            AXIS_10_POSITION : Real;   // AXIS 10 POSITION
            AXIS_11_POSITION : Real;   // AXIS 11 POSITION
            AXIS_12_POSITION : Real;   // AXIS 12 POSITION
            AXIS_13_POSITION : Real;   // AXIS 13 POSITION
            AXIS_14_POSITION : Real;   // AXIS 14 POSITION
            AXIS_15_POSITION : Real;   // AXIS 15 POSITION
            AXIS_16_POSITION : Real;   // AXIS 16 POSITION
            AXIS_17_POSITION : Real;   // AXIS 17 POSITION
            AXIS_18_POSITION : Real;   // AXIS 18 POSITION
            AXIS_19_POSITION : Real;   // AXIS 19 POSITION
            AXIS_20_POSITION : Real;   // AXIS 20 POSITION
            AXIS_21_POSITION : Real;   // AXIS 21 POSITION
            AXIS_22_POSITION : Real;   // AXIS 22 POSITION
            AXIS_23_POSITION : Real;   // AXIS 23 POSITION
            AXIS_24_POSITION : Real;   // AXIS 24 POSITION
            AXIS_25_POSITION : Real;   // AXIS 25 POSITION
            AXIS_26_POSITION : Real;   // AXIS 26 POSITION
            AXIS_27_POSITION : Real;   // AXIS 27 POSITION
            AXIS_28_POSITION : Real;   // AXIS 28 POSITION
            AXIS_29_POSITION : Real;   // AXIS 29 POSITION
            AXIS_30_POSITION : Real;   // AXIS 30 POSITION
            AXIS_31_POSITION : Real;   // AXIS 31 POSITION
         END_STRUCT;
         AUX : Struct
            AUX1 : Bool;   // AUXILIAR 1
            AUX2 : Bool;   // AUXILIAR 2
            AUX3 : Bool;   // AUXILIAR 3
            AUX4 : Bool;   // AUXILIAR 4
            AUX5 : Bool;   // AUXILIAR 5
            AUX6 : Bool;   // AUXILIAR 6
            AUX7 : Bool;   // AUXILIAR 7
            AUX8 : Byte;   // AUXILIAR 8
            AUX9 : Byte;   // AUXILIAR 9
            AUX10 : Byte;   // AUXILIAR 10
            AUX11 : Byte;   // AUXILIAR 11
            AUX12 : Byte;   // AUXILIAR 12
            AUX13 : Byte;   // AUXILIAR 13
            AUX14 : Byte;   // AUXILIAR 14
         END_STRUCT;
         REFERENCE_SCREEN : Struct
            AXIS_SELECTED : Int;   // REFERENCE SCREEN AXIS SELECTED
            MEMO_AXIS_SELECTED : Int;   // REFERENCE SCREEN MEMORIZED AXIS SELECTED
            SCREEN_SELECTED : Bool;   // REFERENCE SCREEN SCREEN SELECTED
            READ_DATA : Bool;   // REFERENCE SCREEN READ DATA
            WRITE_DATA : Bool;   // REFERENCE SCREEN WRITE DATA
            TIMER_READ : TP_TIME;   // READ TIMER
         END_STRUCT;
      END_STRUCT;
      MG7 : Struct
         GENERAL_BITS : Struct
            SCREEN_BA3_SELECTED : Bool;   // SCREEN BA3 SELECTED / GENERAL BITS SCREEN BA3 SELECTED
            SCREEN_NC_MANUAL_SELECTED : Bool;   // SCREEN NC MANUAL SELECTED / GENERAL BITS SCREEN NC MANUAL SELECTED
            SCREEN_EB_MODE_SELECT : Bool;   // SCREEN EB MODE SELECT / GENERAL BITS SCREEN EB MODE SELECT
            SP0_3 : Bool;   // GENERAL BITS
            BA3_SELECTED_UNIT_1 : Bool;   // BA3 SELECTED UNIT 1 / GENERAL BITS BA3 LIST SELECTED UNIT 1
            BA3_SELECTED_UNIT_2 : Bool;   // BA3 SELECTED UNIT 2 / GENERAL BITS BA3 LIST SELECTED UNIT 2
            BA3_SELECTED_UNIT_3 : Bool;   // BA3 SELECTED UNIT 3 / GENERAL BITS BA3 LIST SELECTED UNIT 3
            BA3_SELECTED_UNIT_4 : Bool;   // BA3 SELECTED UNIT 4 / GENERAL BITS BA3 LIST SELECTED UNIT 4
            SP1_0 : Bool;   // TWO UNITS OPTION ENABLE / GENERAL BITS
            SPNDLS_SBH_SG_AUX : Bool;   // GENERAL BITS SPINDLES SBH SG AUX
            SPNDLS_SBH_SG_PULSE : Bool;   // GENERAL BITS SPINDLES SBH SG PULSE
            PLC_LINE_AXES_BYTE : Byte;   // GENERAL BITS PLC LINE AXES BYTE
            PLC_LINE_SPINDLES_BYTE : Byte;   // GENERAL BITS PLC LINE SPINDLES BYTE
            PLC_LINE_AXES : Int;   // GENERAL BITS PLC LINE AXES
            PLC_LINE_SPINDLES : Int;   // GENERAL BITS PLC LINE SPINDLES
            BA3_LIST : Int;   // GENERAL BITS BA3 LIST
            MINUS_KEY : Byte;   // GENERAL BITS MINUS KEY
            PLUS_KEY : Byte;   // GENERAL BITS PLUS KEY
         END_STRUCT;
         NC_AXES : Struct
            SOFTKEYS : Struct   // NC AXES SOFTKEYS
               LEFT : Struct
                  MANUAL_MODE : Bool;   // MANUAL MODE (CN-AXES SCREEN) / NC AXES SOFTKEYS MANUAL MODE
                  SEMIAUTOMATIC_MODE : Bool;   // SEMIAUTOMATIC MODE (CN-AXES SCREEN) / NC AXES SOFTKEYS SEMIAUTOMATIC MODE
                  REFERENCE_MODE : Bool;   // REFERENCE MODE (CN-AXES SCREEN) / NC AXES SOFTKEYS REFERENCE MODE
                  JOG_MODE : Bool;   // NC AXES SOFTKEYS SPARE
                  SPINDLES_SBH_SG : Bool;   // SPINDLES SBH SG (CN-AXES SCREEN) / NC AXES SOFTKEYS SPINDLES SBH SG
                  CONTINUOS_INCREMENTAL : Bool;   // CONTINUOS-INCREMENTAL (CN-AXES SCREEN) / NC AXES SOFTKEYS CONTINUOS INCREMENTAL
                  SP0_6 : Bool;   // NC AXES SOFTKEYS SP0 6
                  SP0_7 : Bool;   // NC AXES SOFTKEYS SP0 7
               END_STRUCT;
               RIGHT : Struct
                  JOG_PLUS : Bool;   // JOG PLUS (CN-AXES SCREEN) / NC AXES SOFTKEYS JOG PLUS
                  JOG_MINUS : Bool;   // JOG MINUS (CN-AXES SCREEN) / NC AXES SOFTKEYS JOG MINUS
                  BLOCK_DEVICE : Bool;   // BLOCK DEVICE (CN-AXES SCREEN) / NC AXES SOFTKEYS BLOCK DEVICE
                  UNBLOCK_DEVICE : Bool;   // UNBLOCK DEVICE (CN-AXES SCREEN) / NC AXES SOFTKEYS UNBLOCK DEVICE
                  SP1_4 : Bool;   // NC AXES SOFTKEYS SP1 4
                  CHANGE_PANEL_CONTROL : Bool;   // CHANGE PANEL CONTROL (CN-AXES SCREEN) / NC AXES SOFTKEYS CHANGE PANEL CONTROL
                  SP1_6 : Bool;   // NC AXES SOFTKEYS SP1 6
                  SP1_7 : Bool;   // NC AXES SOFTKEYS SP1 7
               END_STRUCT;
            END_STRUCT;
            PBS : Struct   // NC AXES PBS
               MICRON : Bool;   // NC AXES PBS MICRON
               MICRONS_10 : Bool;   // NC AXES PBS MICRONS 10
               MICRONS_100 : Bool;   // NC AXES PBS MICRONS 100
               MILIMETER : Bool;   // NC AXES PBS MILIMETER
               SP0_4 : Bool;
               SP0_5 : Bool;
               SP0_6 : Bool;
               SP0_7 : Bool;
               SP1_0 : Bool;
               SP1_1 : Bool;
               SP1_2 : Bool;
               SP1_3 : Bool;
               SP1_4 : Bool;
               SP1_5 : Bool;
               SP1_6 : Bool;
               SP1_7 : Bool;
            END_STRUCT;
            SOFTKEY_LEDS : Struct   // NC AXES SOFTKEY LEDS
               MANUAL_MODE : Bool;   // MANUAL MODE (SOFTKEY LEDS) / NC AXES SOFTKEY LEDS MANUAL MODE
               ES_MODE : Bool;   // NC AXES SOFTKEY LEDS ES MODE
               REFERENCE_MODE : Bool;   // NC AXES SOFTKEY LEDS REFERENCE MODE
               SP0_3 : Bool;   // NC AXES SOFTKEY LEDS SP0 3
               SPINDLES_SBH_SG : Bool;   // NC AXES SOFTKEY LEDS SPINDLES SBH SG
               CONTINUOS_INCREMENTAL : Bool;   // NC AXES SOFTKEY LEDS CONTINUOS INCREMENTAL
               EB_MODE : Bool;   // NC AXES SOFTKEY LEDS EB MODE
               VK_MODE : Bool;   // NC AXES SOFTKEY LEDS VK MODE
               JOG_PLUS : Bool;   // NC AXES SOFTKEY LEDS JOG PLUS
               JOG_MINUS : Bool;   // NC AXES SOFTKEY LEDS JOG MINUS
               BLOCK_DEVICE : Bool;   // NC AXES SOFTKEY LEDS BLOCK DEVICE
               UNBLOCK_DEVICE : Bool;   // NC AXES SOFTKEY LEDS UNBLOCK DEVICE
               SP1_4 : Bool;   // NC AXES SOFTKEY LEDS SP1 4
               CHANGE_PANEL_CONTROL : Bool;   // NC AXES SOFTKEY LEDS CHANGE PANEL CONTROL
               SP1_6 : Bool;   // NC AXES SOFTKEY LEDS SP1 6
               SP1_7 : Bool;   // NC AXES SOFTKEY LEDS SP1 7
            END_STRUCT;
            PBS_LEDS : Struct   // NC AXES PBS LEDS
               MICRON : Bool;   // NC AXES PBS LEDS MICRON
               MICRONS_10 : Bool;   // NC AXES PBS LEDS MICRONS_10
               MICRONS_100 : Bool;   // NC AXES PBS LEDS MICRONS_100
               MILIMETER : Bool;   // NC AXES PBS LEDS MILIMETER
               SP0_4 : Bool;
               SP0_5 : Bool;
               SP0_6 : Bool;
               SP0_7 : Bool;
               SP1_0 : Bool;
               SP1_1 : Bool;
               SP1_2 : Bool;
               SP1_3 : Bool;
               SP1_4 : Bool;
               SP1_5 : Bool;
               SP1_6 : Bool;
               SP1_7 : Bool;
            END_STRUCT;
         END_STRUCT;
         BA3 : Struct
            SOFTKEYS : Struct   // BA3 SOFTKEYS
               AUTOMATIC_MODE : Bool;   // AUTOMATIC MODE (BA3) / BA3 SOFTKEYS AUTOMATIC MODE
               SINGLE_MODE : Bool;   // SINGLE CYCLE MODE (BA3) / BA3 SOFTKEYS SINGLE MODE
               SEMIAUTOMATIC_MODE : Bool;   // SEMIAUTOMATIC MODE (BA3) / BA3 SOFTKEYS SEMIAUTOMATIC MODE
               MANUAL_MODE : Bool;   // MANUAL MODE (BA3) / BA3 SOFTKEYS MANUAL MODE
               START : Bool;   // START (BA3) / BA3 SOFTKEYS START
               STOP : Bool;   // STOP (BA3) / BA3 SOFTKEYS STOP
               SPARE_2 : Bool;   // BA3 SOFTKEYS SP0 6
               SPARE : Bool;   // BA3 SOFTKEYS SP0 7
               SET_GOOD_PART : Bool;   // BA3 SOFTKEYS CLAMP FIXTURE 1
               UNCLAMP_F1 : Bool;   // BA3 SOFTKEYS UNCLAMP FIXTURE 1
               CLAMP_F2 : Bool;   // BA3 SOFTKEYS CLAMP FIXTURE 2
               UNCLAMP_F2 : Bool;   // BA3 SOFTKEYS UNCLAMP FIXTURE 2
               UNBLOCK_DEVICE : Bool;   // BA3 SOFTKEYS UNBLOCK DEVICE
               HOME : Bool;   // HOME (BA3) / BA3 SOFTKEYS HOME
               END_OF_CYCLE : Bool;   // BA3 SOFTKEYS END OF CYCLE
               CHANGE_PANEL_CONTROL : Bool;   // BA3 SOFTKEYS CHANGE PANEL
            END_STRUCT;
            PBS : Struct   // BA3 PBS
               MICRON : Bool;   // BA3 PBS MICRON
               MICRONS_10 : Bool;   // BA3 PBS MICRONS_10
               MICRONS_100 : Bool;   // BA3 PBS MICRONS_100
               MILIMETER : Bool;   // BA3 PBS MILIMETER
               SP0_4 : Bool;
               SP0_5 : Bool;
               SP0_6 : Bool;
               SP0_7 : Bool;
               SP1_0 : Bool;
               SP1_1 : Bool;
               SP1_2 : Bool;
               SP1_3 : Bool;
               SP1_4 : Bool;
               SP1_5 : Bool;
               SP1_6 : Bool;
               SP1_7 : Bool;
            END_STRUCT;
            SOFTKEY_LEDS : Struct   // BA3 SOFTKEY LEDS
               ER_MODE : Bool;   // BA3 SOFTKEY LEDS ER MODE
               ES_MODE : Bool;   // BA3 SOFTKEY LEDS ES MODE
               HOME : Bool;   // BA3 SOFTKEY LEDS HOME
               START : Bool;   // BA3 SOFTKEY LEDS START
               STOP : Bool;   // BA3 SOFTKEY LEDS STOP
               CONTINUOS_INCREMENTAL : Bool;   // BA3 SOFTKEY LEDS CONTINUOS INCREMENTAL
               SP0_6 : Bool;   // BA3 SOFTKEY LEDS SP0 6
               SP0_7 : Bool;   // BA3 SOFTKEY LEDS SP0 7
               JOG_PLUS : Bool;   // BA3 SOFTKEY LEDS JOG PLUS
               JOG_MINUS : Bool;   // BA3 SOFTKEY LEDS JOG MINUS
               UNBLOCK_DEVICE : Bool;   // BA3 SOFTKEY LEDS UNBLOCK DEVICE
               CLAMP_F1 : Bool;   // BA3 SOFTKEY LEDS CLAMP F1
               UNCLAMP_F1 : Bool;   // BA3 SOFTKEY LEDS UNCLAMP F1
               CLAMP_F2 : Bool;   // BA3 SOFTKEY LEDS CLAMP F2
               UNCLAMP_F2 : Bool;   // BA3 SOFTKEY LEDS UNCLAMP F2
               SP1_7 : Bool;   // BA3 SOFTKEY LEDS SP1 7
            END_STRUCT;
            PBS_LEDS : Struct   // BA3 PBS LEDS
               MICRON : Bool;   // BA3 PBS LEDS MICRON
               MICRONS_10 : Bool;   // BA3 PBS LEDS MICRONS_10
               MICRONS_100 : Bool;   // BA3 PBS LEDS MICRONS_100
               MILIMETER : Bool;   // BA3 PBS LEDS MILIMETER
               SP0_4 : Bool;
               SP0_5 : Bool;
               SP0_6 : Bool;
               SP0_7 : Bool;
               SP1_0 : Bool;
               SP1_1 : Bool;
               SP1_2 : Bool;
               SP1_3 : Bool;
               SP1_4 : Bool;
               SP1_5 : Bool;
               SP1_6 : Bool;
               BA3_MODE_SELECTED : Bool;
            END_STRUCT;
         END_STRUCT;
         AXIS_SELECTED : Struct
            AXIS_1_SELECTED : Bool;   // SPINDLE SP11 SELECTED / AXIS 1 SELECTED
            AXIS_2_SELECTED : Bool;   // SPINDLE SP12 SELECTED / AXIS 2 SELECTED
            AXIS_3_SELECTED : Bool;   // SPINDLE SP13 SELECTED / AXIS 3 SELECTED
            AXIS_4_SELECTED : Bool;   // SPINDLE SP14 SELECTED / AXIS 4 SELECTED
            AXIS_5_SELECTED : Bool;   // AXIS X1 SELECTED / AXIS 5 SELECTED
            AXIS_6_SELECTED : Bool;   // AXIS Y1 SELECTED / AXIS 6 SELECTED
            AXIS_7_SELECTED : Bool;   // AXIS Z11 SELECTED / AXIS 7 SELECTED
            AXIS_8_SELECTED : Bool;   // AXIS Z12 SELECTED / AXIS 8 SELECTED
            AXIS_9_SELECTED : Bool;   // AXIS X2 SELECTED / AXIS 9 SELECTED
            AXIS_10_SELECTED : Bool;   // AXIS Y2 SELECTED / AXIS 10 SELECTED
            AXIS_11_SELECTED : Bool;   // AXIS Z21 SELECTED / AXIS 11 SELECTED
            AXIS_12_SELECTED : Bool;   // AXIS Z22 SELECTED / AXIS 12 SELECTED
            AXIS_13_SELECTED : Bool;   // AXIS Q1 SELECTED / AXIS 13 SELECTED
            AXIS_14_SELECTED : Bool;   // AXIS Q2 SELECTED / AXIS 14 SELECTED
            AXIS_15_SELECTED : Bool;   // AXIS A1 SELECTED / AXIS 15 SELECTED
            AXIS_16_SELECTED : Bool;   // AXIS B SELECTED / AXIS 16 SELECTED
            AXIS_17_SELECTED : Bool;   // AXIS W SELECTED / AXIS 17 SELECTED
            AXIS_18_SELECTED : Bool;   // AXIS E SELECTED / AXIS 18 SELECTED
            AXIS_19_SELECTED : Bool;   // AXIS A2 SELECTED / AXIS 19 SELECTED
            AXIS_20_SELECTED : Bool;   // AXIS V1 SELECTED / AXIS 20 SELECTED
            AXIS_21_SELECTED : Bool;   // AXIS V2 SELECTED / AXIS 21 SELECTED
            AXIS_22_SELECTED : Bool;   // AXIS R SELECTED / AXIS 22 SELECTED
            AXIS_23_SELECTED : Bool;   // AXIS U1 SELECTED / AXIS 23 SELECTED
            AXIS_24_SELECTED : Bool;   // AXIS U2 SELECTED / AXIS 24 SELECTED
            AXIS_25_SELECTED : Bool;   // AXIS C SELECTED / AXIS 25 SELECTED
            AXIS_26_SELECTED : Bool;   // AXIS W1 SELECTED / AXIS 26 SELECTED
            AXIS_27_SELECTED : Bool;   // AXIS V SELECTED / AXIS 27 SELECTED
            AXIS_28_SELECTED : Bool;   // AXIS 28 SELECTED
            AXIS_29_SELECTED : Bool;   // AXIS 29 SELECTED
            AXIS_30_SELECTED : Bool;   // AXIS 30 SELECTED
            AXIS_31_SELECTED : Bool;   // AXIS 31 SELECTED
            SPARE_33_7 : Bool;   // SPARE_33_7
         END_STRUCT;
         AXIS_REFERENCED : Struct
            AXIS_1_REFERENCED : Bool;   // SPINDLE SP11 REFERENCED / AXIS 1 REFERENCED
            AXIS_2_REFERENCED : Bool;   // SPINDLE SP12 REFERENCED / AXIS 2 REFERENCED
            AXIS_3_REFERENCED : Bool;   // SPINDLE SP13 REFERENCED / AXIS 3 REFERENCED
            AXIS_4_REFERENCED : Bool;   // SPINDLE SP14 REFERENCED / AXIS 4 REFERENCED
            AXIS_5_REFERENCED : Bool;   // AXIS X1 REFERENCED / AXIS 5 REFERENCED
            AXIS_6_REFERENCED : Bool;   // AXIS Y1 REFERENCED / AXIS 6 REFERENCED
            AXIS_7_REFERENCED : Bool;   // AXIS Z11 REFERENCED / AXIS 7 REFERENCED
            AXIS_8_REFERENCED : Bool;   // AXIS Z12 REFERENCED / AXIS 8 REFERENCED
            AXIS_9_REFERENCED : Bool;   // AXIS X2 REFERENCED / AXIS 9 REFERENCED
            AXIS_10_REFERENCED : Bool;   // AXIS Y2 REFERENCED / AXIS 10 REFERENCED
            AXIS_11_REFERENCED : Bool;   // AXIS Z21 REFERENCED / AXIS 11 REFERENCED
            AXIS_12_REFERENCED : Bool;   // AXIS Z22 REFERENCED / AXIS 12 REFERENCED
            AXIS_13_REFERENCED : Bool;   // AXIS Q1 REFERENCED / AXIS 13 REFERENCED
            AXIS_14_REFERENCED : Bool;   // AXIS Q2 REFERENCED / AXIS 14 REFERENCED
            AXIS_15_REFERENCED : Bool;   // AXIS A1 REFERENCED / AXIS 15 REFERENCED
            AXIS_16_REFERENCED : Bool;   // AXIS B REFERENCED / AXIS 16 REFERENCED
            AXIS_17_REFERENCED : Bool;   // AXIS W REFERENCED / AXIS 17 REFERENCED
            AXIS_18_REFERENCED : Bool;   // AXIS E REFERENCED / AXIS 18 REFERENCED
            AXIS_19_REFERENCED : Bool;   // AXIS A2 REFERENCED / AXIS 19 REFERENCED
            AXIS_20_REFERENCED : Bool;   // AXIS V1 REFERENCED / AXIS 20 REFERENCED
            AXIS_21_REFERENCED : Bool;   // AXIS V2 REFERENCED / AXIS 21 REFERENCED
            AXIS_22_REFERENCED : Bool;   // AXIS R REFERENCED / AXIS 22 REFERENCED
            AXIS_23_REFERENCED : Bool;   // AXIS U1 REFERENCED / AXIS 23 REFERENCED
            AXIS_24_REFERENCED : Bool;   // AXIS U2 REFERENCED / AXIS 24 REFERENCED
            AXIS_25_REFERENCED : Bool;   // AXIS C REFERENCED / AXIS 25 REFERENCED
            AXIS_26_REFERENCED : Bool;   // AXIS W1 REFERENCED / AXIS 26 REFERENCED
            AXIS_27_REFERENCED : Bool;   // AXIS V REFERENCED / AXIS 27 REFERENCED
            AXIS_28_REFERENCED : Bool;   // AXIS 28 REFERENCED
            AXIS_29_REFERENCED : Bool;   // AXIS 29 REFERENCED
            AXIS_30_REFERENCED : Bool;   // AXIS 30 REFERENCED
            AXIS_31_REFERENCED : Bool;   // AXIS 31 REFERENCED
            SPARE_37_7 : Bool;   // SPARE_37_7
         END_STRUCT;
         AXIS_CONDITIONS : Struct
            AXIS_1_CONDITIONS : Bool;   // SPINDLE SP11 CONDITIONS / AXIS 1 CONDITIONS
            AXIS_2_CONDITIONS : Bool;   // SPINDLE SP12 CONDITIONS / AXIS 2 CONDITIONS
            AXIS_3_CONDITIONS : Bool;   // SPINDLE SP13 CONDITIONS / AXIS 3 CONDITIONS
            AXIS_4_CONDITIONS : Bool;   // SPINDLE SP14 CONDITIONS / AXIS 4 CONDITIONS
            AXIS_5_CONDITIONS : Bool;   // AXIS X1 CONDITIONS / AXIS 5 CONDITIONS
            AXIS_6_CONDITIONS : Bool;   // AXIS Y1 CONDITIONS / AXIS 6 CONDITIONS
            AXIS_7_CONDITIONS : Bool;   // AXIS Z11 CONDITIONS / AXIS 7 CONDITIONS
            AXIS_8_CONDITIONS : Bool;   // AXIS Z12 CONDITIONS / AXIS 8 CONDITIONS
            AXIS_9_CONDITIONS : Bool;   // AXIS X2 CONDITIONS / AXIS 9 CONDITIONS
            AXIS_10_CONDITIONS : Bool;   // AXIS Y2 CONDITIONS / AXIS 10 CONDITIONS
            AXIS_11_CONDITIONS : Bool;   // AXIS Z21 CONDITIONS / AXIS 11 CONDITIONS
            AXIS_12_CONDITIONS : Bool;   // AXIS Z22 CONDITIONS / AXIS 12 CONDITIONS
            AXIS_13_CONDITIONS : Bool;   // AXIS Q1 CONDITIONS / AXIS 13 CONDITIONS
            AXIS_14_CONDITIONS : Bool;   // AXIS Q2 CONDITIONS / AXIS 14 CONDITIONS
            AXIS_15_CONDITIONS : Bool;   // AXIS A1 CONDITIONS / AXIS 15 CONDITIONS
            AXIS_16_CONDITIONS : Bool;   // AXIS B CONDITIONS / AXIS 16 CONDITIONS
            AXIS_17_CONDITIONS : Bool;   // AXIS W CONDITIONS / AXIS 17 CONDITIONS
            AXIS_18_CONDITIONS : Bool;   // AXIS E CONDITIONS / AXIS 18 CONDITIONS
            AXIS_19_CONDITIONS : Bool;   // AXIS A2 CONDITIONS / AXIS 19 CONDITIONS
            AXIS_20_CONDITIONS : Bool;   // AXIS V1 CONDITIONS / AXIS 20 CONDITIONS
            AXIS_21_CONDITIONS : Bool;   // AXIS V2 CONDITIONS / AXIS 21 CONDITIONS
            AXIS_22_CONDITIONS : Bool;   // AXIS R CONDITIONS / AXIS 22 CONDITIONS
            AXIS_23_CONDITIONS : Bool;   // AXIS U1 CONDITIONS / AXIS 23 CONDITIONS
            AXIS_24_CONDITIONS : Bool;   // AXIS U2 CONDITIONS / AXIS 24 CONDITIONS
            AXIS_25_CONDITIONS : Bool;   // AXIS C CONDITIONS / AXIS 25 CONDITIONS
            AXIS_26_CONDITIONS : Bool;   // AXIS W1 CONDITIONS / AXIS 26 CONDITIONS
            AXIS_27_CONDITIONS : Bool;   // AXIS V CONDITIONS / AXIS 27 CONDITIONS
            AXIS_28_CONDITIONS : Bool;   // AXIS 28 CONDITIONS
            AXIS_29_CONDITIONS : Bool;   // AXIS 29 CONDITIONS
            AXIS_30_CONDITIONS : Bool;   // AXIS 30 CONDITIONS
            AXIS_31_CONDITIONS : Bool;   // AXIS 31 CONDITIONS
            SPARE_41_7 : Bool;   // SPARE_41_7
         END_STRUCT;
         AXIS_POSITION : Struct
            AXIS_1_POSITION : Real;   // AXIS 1 POSITION
            AXIS_2_POSITION : Real;   // AXIS 2 POSITION
            AXIS_3_POSITION : Real;   // AXIS 3 POSITION
            AXIS_4_POSITION : Real;   // AXIS 4 POSITION
            AXIS_5_POSITION : Real;   // AXIS 5 POSITION
            AXIS_6_POSITION : Real;   // AXIS 6 POSITION
            AXIS_7_POSITION : Real;   // AXIS 7 POSITION
            AXIS_8_POSITION : Real;   // AXIS 8 POSITION
            AXIS_9_POSITION : Real;   // AXIS 9 POSITION
            AXIS_10_POSITION : Real;   // AXIS 10 POSITION
            AXIS_11_POSITION : Real;   // AXIS 11 POSITION
            AXIS_12_POSITION : Real;   // AXIS 12 POSITION
            AXIS_13_POSITION : Real;   // AXIS 13 POSITION
            AXIS_14_POSITION : Real;   // AXIS 14 POSITION
            AXIS_15_POSITION : Real;   // AXIS 15 POSITION
            AXIS_16_POSITION : Real;   // AXIS 16 POSITION
            AXIS_17_POSITION : Real;   // AXIS 17 POSITION
            AXIS_18_POSITION : Real;   // AXIS 18 POSITION
            AXIS_19_POSITION : Real;   // AXIS 19 POSITION
            AXIS_20_POSITION : Real;   // AXIS 20 POSITION
            AXIS_21_POSITION : Real;   // AXIS 21 POSITION
            AXIS_22_POSITION : Real;   // AXIS 22 POSITION
            AXIS_23_POSITION : Real;   // AXIS 23 POSITION
            AXIS_24_POSITION : Real;   // AXIS 24 POSITION
            AXIS_25_POSITION : Real;   // AXIS 25 POSITION
            AXIS_26_POSITION : Real;   // AXIS 26 POSITION
            AXIS_27_POSITION : Real;   // AXIS 27 POSITION
            AXIS_28_POSITION : Real;   // AXIS 28 POSITION
            AXIS_29_POSITION : Real;   // AXIS 29 POSITION
            AXIS_30_POSITION : Real;   // AXIS 30 POSITION
            AXIS_31_POSITION : Real;   // AXIS 31 POSITION
         END_STRUCT;
         AUX : Struct
            AUX1 : Bool;   // AUXILIAR 1
            AUX2 : Bool;   // AUXILIAR 2
            AUX3 : Bool;   // AUXILIAR 3
            AUX4 : Bool;   // AUXILIAR 4
            AUX5 : Bool;   // AUXILIAR 5
            AUX6 : Bool;   // AUXILIAR 6
            AUX7 : Bool;   // AUXILIAR 7
            AUX8 : Byte;   // AUXILIAR 8
            AUX9 : Byte;   // AUXILIAR 9
            AUX10 : Byte;   // AUXILIAR 10
            AUX11 : Byte;   // AUXILIAR 11
            AUX12 : Byte;   // AUXILIAR 12
            AUX13 : Byte;   // AUXILIAR 13
            AUX14 : Byte;   // AUXILIAR 14
         END_STRUCT;
         REFERENCE_SCREEN : Struct
            AXIS_SELECTED : Int;   // REFERENCE SCREEN AXIS SELECTED
            MEMO_AXIS_SELECTED : Int;   // REFERENCE SCREEN MEMORIZED AXIS SELECTED
            SCREEN_SELECTED : Bool;   // REFERENCE SCREEN SCREEN SELECTED
            READ_DATA : Bool;   // REFERENCE SCREEN READ DATA
            WRITE_DATA : Bool;   // REFERENCE SCREEN WRITE DATA
            TIMER_READ : TP_TIME;   // READ TIMER
         END_STRUCT;
      END_STRUCT;
      MG8 : Struct
         GENERAL_BITS : Struct
            SCREEN_BA3_SELECTED : Bool;   // SCREEN BA3 SELECTED / GENERAL BITS SCREEN BA3 SELECTED
            SCREEN_NC_MANUAL_SELECTED : Bool;   // SCREEN NC MANUAL SELECTED / GENERAL BITS SCREEN NC MANUAL SELECTED
            SCREEN_EB_MODE_SELECT : Bool;   // SCREEN EB MODE SELECT / GENERAL BITS SCREEN EB MODE SELECT
            SP0_3 : Bool;   // GENERAL BITS
            BA3_SELECTED_UNIT_1 : Bool;   // BA3 SELECTED UNIT 1 / GENERAL BITS BA3 LIST SELECTED UNIT 1
            BA3_SELECTED_UNIT_2 : Bool;   // BA3 SELECTED UNIT 2 / GENERAL BITS BA3 LIST SELECTED UNIT 2
            BA3_SELECTED_UNIT_3 : Bool;   // BA3 SELECTED UNIT 3 / GENERAL BITS BA3 LIST SELECTED UNIT 3
            BA3_SELECTED_UNIT_4 : Bool;   // BA3 SELECTED UNIT 4 / GENERAL BITS BA3 LIST SELECTED UNIT 4
            SP1_0 : Bool;   // TWO UNITS OPTION ENABLE / GENERAL BITS
            SPNDLS_SBH_SG_AUX : Bool;   // GENERAL BITS SPINDLES SBH SG AUX
            SPNDLS_SBH_SG_PULSE : Bool;   // GENERAL BITS SPINDLES SBH SG PULSE
            PLC_LINE_AXES_BYTE : Byte;   // GENERAL BITS PLC LINE AXES BYTE
            PLC_LINE_SPINDLES_BYTE : Byte;   // GENERAL BITS PLC LINE SPINDLES BYTE
            PLC_LINE_AXES : Int;   // GENERAL BITS PLC LINE AXES
            PLC_LINE_SPINDLES : Int;   // GENERAL BITS PLC LINE SPINDLES
            BA3_LIST : Int;   // GENERAL BITS BA3 LIST
            MINUS_KEY : Byte;   // GENERAL BITS MINUS KEY
            PLUS_KEY : Byte;   // GENERAL BITS PLUS KEY
         END_STRUCT;
         NC_AXES : Struct
            SOFTKEYS : Struct   // NC AXES SOFTKEYS
               LEFT : Struct
                  MANUAL_MODE : Bool;   // MANUAL MODE (CN-AXES SCREEN) / NC AXES SOFTKEYS MANUAL MODE
                  SEMIAUTOMATIC_MODE : Bool;   // SEMIAUTOMATIC MODE (CN-AXES SCREEN) / NC AXES SOFTKEYS SEMIAUTOMATIC MODE
                  REFERENCE_MODE : Bool;   // REFERENCE MODE (CN-AXES SCREEN) / NC AXES SOFTKEYS REFERENCE MODE
                  JOG_MODE : Bool;   // NC AXES SOFTKEYS SPARE
                  SPINDLES_SBH_SG : Bool;   // SPINDLES SBH SG (CN-AXES SCREEN) / NC AXES SOFTKEYS SPINDLES SBH SG
                  CONTINUOS_INCREMENTAL : Bool;   // CONTINUOS-INCREMENTAL (CN-AXES SCREEN) / NC AXES SOFTKEYS CONTINUOS INCREMENTAL
                  SP0_6 : Bool;   // NC AXES SOFTKEYS SP0 6
                  SP0_7 : Bool;   // NC AXES SOFTKEYS SP0 7
               END_STRUCT;
               RIGHT : Struct
                  JOG_PLUS : Bool;   // JOG PLUS (CN-AXES SCREEN) / NC AXES SOFTKEYS JOG PLUS
                  JOG_MINUS : Bool;   // JOG MINUS (CN-AXES SCREEN) / NC AXES SOFTKEYS JOG MINUS
                  BLOCK_DEVICE : Bool;   // BLOCK DEVICE (CN-AXES SCREEN) / NC AXES SOFTKEYS BLOCK DEVICE
                  UNBLOCK_DEVICE : Bool;   // UNBLOCK DEVICE (CN-AXES SCREEN) / NC AXES SOFTKEYS UNBLOCK DEVICE
                  SP1_4 : Bool;   // NC AXES SOFTKEYS SP1 4
                  CHANGE_PANEL_CONTROL : Bool;   // CHANGE PANEL CONTROL (CN-AXES SCREEN) / NC AXES SOFTKEYS CHANGE PANEL CONTROL
                  SP1_6 : Bool;   // NC AXES SOFTKEYS SP1 6
                  SP1_7 : Bool;   // NC AXES SOFTKEYS SP1 7
               END_STRUCT;
            END_STRUCT;
            PBS : Struct   // NC AXES PBS
               MICRON : Bool;   // NC AXES PBS MICRON
               MICRONS_10 : Bool;   // NC AXES PBS MICRONS 10
               MICRONS_100 : Bool;   // NC AXES PBS MICRONS 100
               MILIMETER : Bool;   // NC AXES PBS MILIMETER
               SP0_4 : Bool;
               SP0_5 : Bool;
               SP0_6 : Bool;
               SP0_7 : Bool;
               SP1_0 : Bool;
               SP1_1 : Bool;
               SP1_2 : Bool;
               SP1_3 : Bool;
               SP1_4 : Bool;
               SP1_5 : Bool;
               SP1_6 : Bool;
               SP1_7 : Bool;
            END_STRUCT;
            SOFTKEY_LEDS : Struct   // NC AXES SOFTKEY LEDS
               MANUAL_MODE : Bool;   // MANUAL MODE (SOFTKEY LEDS) / NC AXES SOFTKEY LEDS MANUAL MODE
               ES_MODE : Bool;   // NC AXES SOFTKEY LEDS ES MODE
               REFERENCE_MODE : Bool;   // NC AXES SOFTKEY LEDS REFERENCE MODE
               SP0_3 : Bool;   // NC AXES SOFTKEY LEDS SP0 3
               SPINDLES_SBH_SG : Bool;   // NC AXES SOFTKEY LEDS SPINDLES SBH SG
               CONTINUOS_INCREMENTAL : Bool;   // NC AXES SOFTKEY LEDS CONTINUOS INCREMENTAL
               EB_MODE : Bool;   // NC AXES SOFTKEY LEDS EB MODE
               VK_MODE : Bool;   // NC AXES SOFTKEY LEDS VK MODE
               JOG_PLUS : Bool;   // NC AXES SOFTKEY LEDS JOG PLUS
               JOG_MINUS : Bool;   // NC AXES SOFTKEY LEDS JOG MINUS
               BLOCK_DEVICE : Bool;   // NC AXES SOFTKEY LEDS BLOCK DEVICE
               UNBLOCK_DEVICE : Bool;   // NC AXES SOFTKEY LEDS UNBLOCK DEVICE
               SP1_4 : Bool;   // NC AXES SOFTKEY LEDS SP1 4
               CHANGE_PANEL_CONTROL : Bool;   // NC AXES SOFTKEY LEDS CHANGE PANEL CONTROL
               SP1_6 : Bool;   // NC AXES SOFTKEY LEDS SP1 6
               SP1_7 : Bool;   // NC AXES SOFTKEY LEDS SP1 7
            END_STRUCT;
            PBS_LEDS : Struct   // NC AXES PBS LEDS
               MICRON : Bool;   // NC AXES PBS LEDS MICRON
               MICRONS_10 : Bool;   // NC AXES PBS LEDS MICRONS_10
               MICRONS_100 : Bool;   // NC AXES PBS LEDS MICRONS_100
               MILIMETER : Bool;   // NC AXES PBS LEDS MILIMETER
               SP0_4 : Bool;
               SP0_5 : Bool;
               SP0_6 : Bool;
               SP0_7 : Bool;
               SP1_0 : Bool;
               SP1_1 : Bool;
               SP1_2 : Bool;
               SP1_3 : Bool;
               SP1_4 : Bool;
               SP1_5 : Bool;
               SP1_6 : Bool;
               SP1_7 : Bool;
            END_STRUCT;
         END_STRUCT;
         BA3 : Struct
            SOFTKEYS : Struct   // BA3 SOFTKEYS
               AUTOMATIC_MODE : Bool;   // AUTOMATIC MODE (BA3) / BA3 SOFTKEYS AUTOMATIC MODE
               SINGLE_MODE : Bool;   // SINGLE CYCLE MODE (BA3) / BA3 SOFTKEYS SINGLE MODE
               SEMIAUTOMATIC_MODE : Bool;   // SEMIAUTOMATIC MODE (BA3) / BA3 SOFTKEYS SEMIAUTOMATIC MODE
               MANUAL_MODE : Bool;   // MANUAL MODE (BA3) / BA3 SOFTKEYS MANUAL MODE
               START : Bool;   // START (BA3) / BA3 SOFTKEYS START
               STOP : Bool;   // STOP (BA3) / BA3 SOFTKEYS STOP
               SPARE_2 : Bool;   // BA3 SOFTKEYS SP0 6
               SPARE : Bool;   // BA3 SOFTKEYS SP0 7
               SET_GOOD_PART : Bool;   // BA3 SOFTKEYS CLAMP FIXTURE 1
               UNCLAMP_F1 : Bool;   // BA3 SOFTKEYS UNCLAMP FIXTURE 1
               CLAMP_F2 : Bool;   // BA3 SOFTKEYS CLAMP FIXTURE 2
               UNCLAMP_F2 : Bool;   // BA3 SOFTKEYS UNCLAMP FIXTURE 2
               UNBLOCK_DEVICE : Bool;   // BA3 SOFTKEYS UNBLOCK DEVICE
               HOME : Bool;   // HOME (BA3) / BA3 SOFTKEYS HOME
               END_OF_CYCLE : Bool;   // BA3 SOFTKEYS END OF CYCLE
               CHANGE_PANEL_CONTROL : Bool;   // BA3 SOFTKEYS CHANGE PANEL
            END_STRUCT;
            PBS : Struct   // BA3 PBS
               MICRON : Bool;   // BA3 PBS MICRON
               MICRONS_10 : Bool;   // BA3 PBS MICRONS_10
               MICRONS_100 : Bool;   // BA3 PBS MICRONS_100
               MILIMETER : Bool;   // BA3 PBS MILIMETER
               SP0_4 : Bool;
               SP0_5 : Bool;
               SP0_6 : Bool;
               SP0_7 : Bool;
               SP1_0 : Bool;
               SP1_1 : Bool;
               SP1_2 : Bool;
               SP1_3 : Bool;
               SP1_4 : Bool;
               SP1_5 : Bool;
               SP1_6 : Bool;
               SP1_7 : Bool;
            END_STRUCT;
            SOFTKEY_LEDS : Struct   // BA3 SOFTKEY LEDS
               ER_MODE : Bool;   // BA3 SOFTKEY LEDS ER MODE
               ES_MODE : Bool;   // BA3 SOFTKEY LEDS ES MODE
               HOME : Bool;   // BA3 SOFTKEY LEDS HOME
               START : Bool;   // BA3 SOFTKEY LEDS START
               STOP : Bool;   // BA3 SOFTKEY LEDS STOP
               CONTINUOS_INCREMENTAL : Bool;   // BA3 SOFTKEY LEDS CONTINUOS INCREMENTAL
               SP0_6 : Bool;   // BA3 SOFTKEY LEDS SP0 6
               SP0_7 : Bool;   // BA3 SOFTKEY LEDS SP0 7
               JOG_PLUS : Bool;   // BA3 SOFTKEY LEDS JOG PLUS
               JOG_MINUS : Bool;   // BA3 SOFTKEY LEDS JOG MINUS
               UNBLOCK_DEVICE : Bool;   // BA3 SOFTKEY LEDS UNBLOCK DEVICE
               CLAMP_F1 : Bool;   // BA3 SOFTKEY LEDS CLAMP F1
               UNCLAMP_F1 : Bool;   // BA3 SOFTKEY LEDS UNCLAMP F1
               CLAMP_F2 : Bool;   // BA3 SOFTKEY LEDS CLAMP F2
               UNCLAMP_F2 : Bool;   // BA3 SOFTKEY LEDS UNCLAMP F2
               SP1_7 : Bool;   // BA3 SOFTKEY LEDS SP1 7
            END_STRUCT;
            PBS_LEDS : Struct   // BA3 PBS LEDS
               MICRON : Bool;   // BA3 PBS LEDS MICRON
               MICRONS_10 : Bool;   // BA3 PBS LEDS MICRONS_10
               MICRONS_100 : Bool;   // BA3 PBS LEDS MICRONS_100
               MILIMETER : Bool;   // BA3 PBS LEDS MILIMETER
               SP0_4 : Bool;
               SP0_5 : Bool;
               SP0_6 : Bool;
               SP0_7 : Bool;
               SP1_0 : Bool;
               SP1_1 : Bool;
               SP1_2 : Bool;
               SP1_3 : Bool;
               SP1_4 : Bool;
               SP1_5 : Bool;
               SP1_6 : Bool;
               BA3_MODE_SELECTED : Bool;
            END_STRUCT;
         END_STRUCT;
         AXIS_SELECTED : Struct
            AXIS_1_SELECTED : Bool;   // SPINDLE SP11 SELECTED / AXIS 1 SELECTED
            AXIS_2_SELECTED : Bool;   // SPINDLE SP12 SELECTED / AXIS 2 SELECTED
            AXIS_3_SELECTED : Bool;   // SPINDLE SP13 SELECTED / AXIS 3 SELECTED
            AXIS_4_SELECTED : Bool;   // SPINDLE SP14 SELECTED / AXIS 4 SELECTED
            AXIS_5_SELECTED : Bool;   // AXIS X1 SELECTED / AXIS 5 SELECTED
            AXIS_6_SELECTED : Bool;   // AXIS Y1 SELECTED / AXIS 6 SELECTED
            AXIS_7_SELECTED : Bool;   // AXIS Z11 SELECTED / AXIS 7 SELECTED
            AXIS_8_SELECTED : Bool;   // AXIS Z12 SELECTED / AXIS 8 SELECTED
            AXIS_9_SELECTED : Bool;   // AXIS X2 SELECTED / AXIS 9 SELECTED
            AXIS_10_SELECTED : Bool;   // AXIS Y2 SELECTED / AXIS 10 SELECTED
            AXIS_11_SELECTED : Bool;   // AXIS Z21 SELECTED / AXIS 11 SELECTED
            AXIS_12_SELECTED : Bool;   // AXIS Z22 SELECTED / AXIS 12 SELECTED
            AXIS_13_SELECTED : Bool;   // AXIS Q1 SELECTED / AXIS 13 SELECTED
            AXIS_14_SELECTED : Bool;   // AXIS Q2 SELECTED / AXIS 14 SELECTED
            AXIS_15_SELECTED : Bool;   // AXIS A1 SELECTED / AXIS 15 SELECTED
            AXIS_16_SELECTED : Bool;   // AXIS B SELECTED / AXIS 16 SELECTED
            AXIS_17_SELECTED : Bool;   // AXIS W SELECTED / AXIS 17 SELECTED
            AXIS_18_SELECTED : Bool;   // AXIS E SELECTED / AXIS 18 SELECTED
            AXIS_19_SELECTED : Bool;   // AXIS A2 SELECTED / AXIS 19 SELECTED
            AXIS_20_SELECTED : Bool;   // AXIS V1 SELECTED / AXIS 20 SELECTED
            AXIS_21_SELECTED : Bool;   // AXIS V2 SELECTED / AXIS 21 SELECTED
            AXIS_22_SELECTED : Bool;   // AXIS R SELECTED / AXIS 22 SELECTED
            AXIS_23_SELECTED : Bool;   // AXIS U1 SELECTED / AXIS 23 SELECTED
            AXIS_24_SELECTED : Bool;   // AXIS U2 SELECTED / AXIS 24 SELECTED
            AXIS_25_SELECTED : Bool;   // AXIS C SELECTED / AXIS 25 SELECTED
            AXIS_26_SELECTED : Bool;   // AXIS W1 SELECTED / AXIS 26 SELECTED
            AXIS_27_SELECTED : Bool;   // AXIS V SELECTED / AXIS 27 SELECTED
            AXIS_28_SELECTED : Bool;   // AXIS 28 SELECTED
            AXIS_29_SELECTED : Bool;   // AXIS 29 SELECTED
            AXIS_30_SELECTED : Bool;   // AXIS 30 SELECTED
            AXIS_31_SELECTED : Bool;   // AXIS 31 SELECTED
            SPARE_33_7 : Bool;   // SPARE_33_7
         END_STRUCT;
         AXIS_REFERENCED : Struct
            AXIS_1_REFERENCED : Bool;   // SPINDLE SP11 REFERENCED / AXIS 1 REFERENCED
            AXIS_2_REFERENCED : Bool;   // SPINDLE SP12 REFERENCED / AXIS 2 REFERENCED
            AXIS_3_REFERENCED : Bool;   // SPINDLE SP13 REFERENCED / AXIS 3 REFERENCED
            AXIS_4_REFERENCED : Bool;   // SPINDLE SP14 REFERENCED / AXIS 4 REFERENCED
            AXIS_5_REFERENCED : Bool;   // AXIS X1 REFERENCED / AXIS 5 REFERENCED
            AXIS_6_REFERENCED : Bool;   // AXIS Y1 REFERENCED / AXIS 6 REFERENCED
            AXIS_7_REFERENCED : Bool;   // AXIS Z11 REFERENCED / AXIS 7 REFERENCED
            AXIS_8_REFERENCED : Bool;   // AXIS Z12 REFERENCED / AXIS 8 REFERENCED
            AXIS_9_REFERENCED : Bool;   // AXIS X2 REFERENCED / AXIS 9 REFERENCED
            AXIS_10_REFERENCED : Bool;   // AXIS Y2 REFERENCED / AXIS 10 REFERENCED
            AXIS_11_REFERENCED : Bool;   // AXIS Z21 REFERENCED / AXIS 11 REFERENCED
            AXIS_12_REFERENCED : Bool;   // AXIS Z22 REFERENCED / AXIS 12 REFERENCED
            AXIS_13_REFERENCED : Bool;   // AXIS Q1 REFERENCED / AXIS 13 REFERENCED
            AXIS_14_REFERENCED : Bool;   // AXIS Q2 REFERENCED / AXIS 14 REFERENCED
            AXIS_15_REFERENCED : Bool;   // AXIS A1 REFERENCED / AXIS 15 REFERENCED
            AXIS_16_REFERENCED : Bool;   // AXIS B REFERENCED / AXIS 16 REFERENCED
            AXIS_17_REFERENCED : Bool;   // AXIS W REFERENCED / AXIS 17 REFERENCED
            AXIS_18_REFERENCED : Bool;   // AXIS E REFERENCED / AXIS 18 REFERENCED
            AXIS_19_REFERENCED : Bool;   // AXIS A2 REFERENCED / AXIS 19 REFERENCED
            AXIS_20_REFERENCED : Bool;   // AXIS V1 REFERENCED / AXIS 20 REFERENCED
            AXIS_21_REFERENCED : Bool;   // AXIS V2 REFERENCED / AXIS 21 REFERENCED
            AXIS_22_REFERENCED : Bool;   // AXIS R REFERENCED / AXIS 22 REFERENCED
            AXIS_23_REFERENCED : Bool;   // AXIS U1 REFERENCED / AXIS 23 REFERENCED
            AXIS_24_REFERENCED : Bool;   // AXIS U2 REFERENCED / AXIS 24 REFERENCED
            AXIS_25_REFERENCED : Bool;   // AXIS C REFERENCED / AXIS 25 REFERENCED
            AXIS_26_REFERENCED : Bool;   // AXIS W1 REFERENCED / AXIS 26 REFERENCED
            AXIS_27_REFERENCED : Bool;   // AXIS V REFERENCED / AXIS 27 REFERENCED
            AXIS_28_REFERENCED : Bool;   // AXIS 28 REFERENCED
            AXIS_29_REFERENCED : Bool;   // AXIS 29 REFERENCED
            AXIS_30_REFERENCED : Bool;   // AXIS 30 REFERENCED
            AXIS_31_REFERENCED : Bool;   // AXIS 31 REFERENCED
            SPARE_37_7 : Bool;   // SPARE_37_7
         END_STRUCT;
         AXIS_CONDITIONS : Struct
            AXIS_1_CONDITIONS : Bool;   // SPINDLE SP11 CONDITIONS / AXIS 1 CONDITIONS
            AXIS_2_CONDITIONS : Bool;   // SPINDLE SP12 CONDITIONS / AXIS 2 CONDITIONS
            AXIS_3_CONDITIONS : Bool;   // SPINDLE SP13 CONDITIONS / AXIS 3 CONDITIONS
            AXIS_4_CONDITIONS : Bool;   // SPINDLE SP14 CONDITIONS / AXIS 4 CONDITIONS
            AXIS_5_CONDITIONS : Bool;   // AXIS X1 CONDITIONS / AXIS 5 CONDITIONS
            AXIS_6_CONDITIONS : Bool;   // AXIS Y1 CONDITIONS / AXIS 6 CONDITIONS
            AXIS_7_CONDITIONS : Bool;   // AXIS Z11 CONDITIONS / AXIS 7 CONDITIONS
            AXIS_8_CONDITIONS : Bool;   // AXIS Z12 CONDITIONS / AXIS 8 CONDITIONS
            AXIS_9_CONDITIONS : Bool;   // AXIS X2 CONDITIONS / AXIS 9 CONDITIONS
            AXIS_10_CONDITIONS : Bool;   // AXIS Y2 CONDITIONS / AXIS 10 CONDITIONS
            AXIS_11_CONDITIONS : Bool;   // AXIS Z21 CONDITIONS / AXIS 11 CONDITIONS
            AXIS_12_CONDITIONS : Bool;   // AXIS Z22 CONDITIONS / AXIS 12 CONDITIONS
            AXIS_13_CONDITIONS : Bool;   // AXIS Q1 CONDITIONS / AXIS 13 CONDITIONS
            AXIS_14_CONDITIONS : Bool;   // AXIS Q2 CONDITIONS / AXIS 14 CONDITIONS
            AXIS_15_CONDITIONS : Bool;   // AXIS A1 CONDITIONS / AXIS 15 CONDITIONS
            AXIS_16_CONDITIONS : Bool;   // AXIS B CONDITIONS / AXIS 16 CONDITIONS
            AXIS_17_CONDITIONS : Bool;   // AXIS W CONDITIONS / AXIS 17 CONDITIONS
            AXIS_18_CONDITIONS : Bool;   // AXIS E CONDITIONS / AXIS 18 CONDITIONS
            AXIS_19_CONDITIONS : Bool;   // AXIS A2 CONDITIONS / AXIS 19 CONDITIONS
            AXIS_20_CONDITIONS : Bool;   // AXIS V1 CONDITIONS / AXIS 20 CONDITIONS
            AXIS_21_CONDITIONS : Bool;   // AXIS V2 CONDITIONS / AXIS 21 CONDITIONS
            AXIS_22_CONDITIONS : Bool;   // AXIS R CONDITIONS / AXIS 22 CONDITIONS
            AXIS_23_CONDITIONS : Bool;   // AXIS U1 CONDITIONS / AXIS 23 CONDITIONS
            AXIS_24_CONDITIONS : Bool;   // AXIS U2 CONDITIONS / AXIS 24 CONDITIONS
            AXIS_25_CONDITIONS : Bool;   // AXIS C CONDITIONS / AXIS 25 CONDITIONS
            AXIS_26_CONDITIONS : Bool;   // AXIS W1 CONDITIONS / AXIS 26 CONDITIONS
            AXIS_27_CONDITIONS : Bool;   // AXIS V CONDITIONS / AXIS 27 CONDITIONS
            AXIS_28_CONDITIONS : Bool;   // AXIS 28 CONDITIONS
            AXIS_29_CONDITIONS : Bool;   // AXIS 29 CONDITIONS
            AXIS_30_CONDITIONS : Bool;   // AXIS 30 CONDITIONS
            AXIS_31_CONDITIONS : Bool;   // AXIS 31 CONDITIONS
            SPARE_41_7 : Bool;   // SPARE_41_7
         END_STRUCT;
         AXIS_POSITION : Struct
            AXIS_1_POSITION : Real;   // AXIS 1 POSITION
            AXIS_2_POSITION : Real;   // AXIS 2 POSITION
            AXIS_3_POSITION : Real;   // AXIS 3 POSITION
            AXIS_4_POSITION : Real;   // AXIS 4 POSITION
            AXIS_5_POSITION : Real;   // AXIS 5 POSITION
            AXIS_6_POSITION : Real;   // AXIS 6 POSITION
            AXIS_7_POSITION : Real;   // AXIS 7 POSITION
            AXIS_8_POSITION : Real;   // AXIS 8 POSITION
            AXIS_9_POSITION : Real;   // AXIS 9 POSITION
            AXIS_10_POSITION : Real;   // AXIS 10 POSITION
            AXIS_11_POSITION : Real;   // AXIS 11 POSITION
            AXIS_12_POSITION : Real;   // AXIS 12 POSITION
            AXIS_13_POSITION : Real;   // AXIS 13 POSITION
            AXIS_14_POSITION : Real;   // AXIS 14 POSITION
            AXIS_15_POSITION : Real;   // AXIS 15 POSITION
            AXIS_16_POSITION : Real;   // AXIS 16 POSITION
            AXIS_17_POSITION : Real;   // AXIS 17 POSITION
            AXIS_18_POSITION : Real;   // AXIS 18 POSITION
            AXIS_19_POSITION : Real;   // AXIS 19 POSITION
            AXIS_20_POSITION : Real;   // AXIS 20 POSITION
            AXIS_21_POSITION : Real;   // AXIS 21 POSITION
            AXIS_22_POSITION : Real;   // AXIS 22 POSITION
            AXIS_23_POSITION : Real;   // AXIS 23 POSITION
            AXIS_24_POSITION : Real;   // AXIS 24 POSITION
            AXIS_25_POSITION : Real;   // AXIS 25 POSITION
            AXIS_26_POSITION : Real;   // AXIS 26 POSITION
            AXIS_27_POSITION : Real;   // AXIS 27 POSITION
            AXIS_28_POSITION : Real;   // AXIS 28 POSITION
            AXIS_29_POSITION : Real;   // AXIS 29 POSITION
            AXIS_30_POSITION : Real;   // AXIS 30 POSITION
            AXIS_31_POSITION : Real;   // AXIS 31 POSITION
         END_STRUCT;
         AUX : Struct
            AUX1 : Bool;   // AUXILIAR 1
            AUX2 : Bool;   // AUXILIAR 2
            AUX3 : Bool;   // AUXILIAR 3
            AUX4 : Bool;   // AUXILIAR 4
            AUX5 : Bool;   // AUXILIAR 5
            AUX6 : Bool;   // AUXILIAR 6
            AUX7 : Bool;   // AUXILIAR 7
            AUX8 : Byte;   // AUXILIAR 8
            AUX9 : Byte;   // AUXILIAR 9
            AUX10 : Byte;   // AUXILIAR 10
            AUX11 : Byte;   // AUXILIAR 11
            AUX12 : Byte;   // AUXILIAR 12
            AUX13 : Byte;   // AUXILIAR 13
            AUX14 : Byte;   // AUXILIAR 14
         END_STRUCT;
         REFERENCE_SCREEN : Struct
            AXIS_SELECTED : Int;   // REFERENCE SCREEN AXIS SELECTED
            MEMO_AXIS_SELECTED : Int;   // REFERENCE SCREEN MEMORIZED AXIS SELECTED
            SCREEN_SELECTED : Bool;   // REFERENCE SCREEN SCREEN SELECTED
            READ_DATA : Bool;   // REFERENCE SCREEN READ DATA
            WRITE_DATA : Bool;   // REFERENCE SCREEN WRITE DATA
            TIMER_READ : TP_TIME;   // READ TIMER
         END_STRUCT;
      END_STRUCT;
      MG9 : Struct
         GENERAL_BITS : Struct
            SCREEN_BA3_SELECTED : Bool;   // SCREEN BA3 SELECTED / GENERAL BITS SCREEN BA3 SELECTED
            SCREEN_NC_MANUAL_SELECTED : Bool;   // SCREEN NC MANUAL SELECTED / GENERAL BITS SCREEN NC MANUAL SELECTED
            SCREEN_EB_MODE_SELECT : Bool;   // SCREEN EB MODE SELECT / GENERAL BITS SCREEN EB MODE SELECT
            SP0_3 : Bool;   // GENERAL BITS
            BA3_SELECTED_UNIT_1 : Bool;   // BA3 SELECTED UNIT 1 / GENERAL BITS BA3 LIST SELECTED UNIT 1
            BA3_SELECTED_UNIT_2 : Bool;   // BA3 SELECTED UNIT 2 / GENERAL BITS BA3 LIST SELECTED UNIT 2
            BA3_SELECTED_UNIT_3 : Bool;   // BA3 SELECTED UNIT 3 / GENERAL BITS BA3 LIST SELECTED UNIT 3
            BA3_SELECTED_UNIT_4 : Bool;   // BA3 SELECTED UNIT 4 / GENERAL BITS BA3 LIST SELECTED UNIT 4
            SP1_0 : Bool;   // TWO UNITS OPTION ENABLE / GENERAL BITS
            SPNDLS_SBH_SG_AUX : Bool;   // GENERAL BITS SPINDLES SBH SG AUX
            SPNDLS_SBH_SG_PULSE : Bool;   // GENERAL BITS SPINDLES SBH SG PULSE
            PLC_LINE_AXES_BYTE : Byte;   // GENERAL BITS PLC LINE AXES BYTE
            PLC_LINE_SPINDLES_BYTE : Byte;   // GENERAL BITS PLC LINE SPINDLES BYTE
            PLC_LINE_AXES : Int;   // GENERAL BITS PLC LINE AXES
            PLC_LINE_SPINDLES : Int;   // GENERAL BITS PLC LINE SPINDLES
            BA3_LIST : Int;   // GENERAL BITS BA3 LIST
            MINUS_KEY : Byte;   // GENERAL BITS MINUS KEY
            PLUS_KEY : Byte;   // GENERAL BITS PLUS KEY
         END_STRUCT;
         NC_AXES : Struct
            SOFTKEYS : Struct   // NC AXES SOFTKEYS
               LEFT : Struct
                  MANUAL_MODE : Bool;   // MANUAL MODE (CN-AXES SCREEN) / NC AXES SOFTKEYS MANUAL MODE
                  SEMIAUTOMATIC_MODE : Bool;   // SEMIAUTOMATIC MODE (CN-AXES SCREEN) / NC AXES SOFTKEYS SEMIAUTOMATIC MODE
                  REFERENCE_MODE : Bool;   // REFERENCE MODE (CN-AXES SCREEN) / NC AXES SOFTKEYS REFERENCE MODE
                  JOG_MODE : Bool;   // NC AXES SOFTKEYS SPARE
                  SPINDLES_SBH_SG : Bool;   // SPINDLES SBH SG (CN-AXES SCREEN) / NC AXES SOFTKEYS SPINDLES SBH SG
                  CONTINUOS_INCREMENTAL : Bool;   // CONTINUOS-INCREMENTAL (CN-AXES SCREEN) / NC AXES SOFTKEYS CONTINUOS INCREMENTAL
                  SP0_6 : Bool;   // NC AXES SOFTKEYS SP0 6
                  SP0_7 : Bool;   // NC AXES SOFTKEYS SP0 7
               END_STRUCT;
               RIGHT : Struct
                  JOG_PLUS : Bool;   // JOG PLUS (CN-AXES SCREEN) / NC AXES SOFTKEYS JOG PLUS
                  JOG_MINUS : Bool;   // JOG MINUS (CN-AXES SCREEN) / NC AXES SOFTKEYS JOG MINUS
                  BLOCK_DEVICE : Bool;   // BLOCK DEVICE (CN-AXES SCREEN) / NC AXES SOFTKEYS BLOCK DEVICE
                  UNBLOCK_DEVICE : Bool;   // UNBLOCK DEVICE (CN-AXES SCREEN) / NC AXES SOFTKEYS UNBLOCK DEVICE
                  SP1_4 : Bool;   // NC AXES SOFTKEYS SP1 4
                  CHANGE_PANEL_CONTROL : Bool;   // CHANGE PANEL CONTROL (CN-AXES SCREEN) / NC AXES SOFTKEYS CHANGE PANEL CONTROL
                  SP1_6 : Bool;   // NC AXES SOFTKEYS SP1 6
                  SP1_7 : Bool;   // NC AXES SOFTKEYS SP1 7
               END_STRUCT;
            END_STRUCT;
            PBS : Struct   // NC AXES PBS
               MICRON : Bool;   // NC AXES PBS MICRON
               MICRONS_10 : Bool;   // NC AXES PBS MICRONS 10
               MICRONS_100 : Bool;   // NC AXES PBS MICRONS 100
               MILIMETER : Bool;   // NC AXES PBS MILIMETER
               SP0_4 : Bool;
               SP0_5 : Bool;
               SP0_6 : Bool;
               SP0_7 : Bool;
               SP1_0 : Bool;
               SP1_1 : Bool;
               SP1_2 : Bool;
               SP1_3 : Bool;
               SP1_4 : Bool;
               SP1_5 : Bool;
               SP1_6 : Bool;
               SP1_7 : Bool;
            END_STRUCT;
            SOFTKEY_LEDS : Struct   // NC AXES SOFTKEY LEDS
               MANUAL_MODE : Bool;   // MANUAL MODE (SOFTKEY LEDS) / NC AXES SOFTKEY LEDS MANUAL MODE
               ES_MODE : Bool;   // NC AXES SOFTKEY LEDS ES MODE
               REFERENCE_MODE : Bool;   // NC AXES SOFTKEY LEDS REFERENCE MODE
               SP0_3 : Bool;   // NC AXES SOFTKEY LEDS SP0 3
               SPINDLES_SBH_SG : Bool;   // NC AXES SOFTKEY LEDS SPINDLES SBH SG
               CONTINUOS_INCREMENTAL : Bool;   // NC AXES SOFTKEY LEDS CONTINUOS INCREMENTAL
               EB_MODE : Bool;   // NC AXES SOFTKEY LEDS EB MODE
               VK_MODE : Bool;   // NC AXES SOFTKEY LEDS VK MODE
               JOG_PLUS : Bool;   // NC AXES SOFTKEY LEDS JOG PLUS
               JOG_MINUS : Bool;   // NC AXES SOFTKEY LEDS JOG MINUS
               BLOCK_DEVICE : Bool;   // NC AXES SOFTKEY LEDS BLOCK DEVICE
               UNBLOCK_DEVICE : Bool;   // NC AXES SOFTKEY LEDS UNBLOCK DEVICE
               SP1_4 : Bool;   // NC AXES SOFTKEY LEDS SP1 4
               CHANGE_PANEL_CONTROL : Bool;   // NC AXES SOFTKEY LEDS CHANGE PANEL CONTROL
               SP1_6 : Bool;   // NC AXES SOFTKEY LEDS SP1 6
               SP1_7 : Bool;   // NC AXES SOFTKEY LEDS SP1 7
            END_STRUCT;
            PBS_LEDS : Struct   // NC AXES PBS LEDS
               MICRON : Bool;   // NC AXES PBS LEDS MICRON
               MICRONS_10 : Bool;   // NC AXES PBS LEDS MICRONS_10
               MICRONS_100 : Bool;   // NC AXES PBS LEDS MICRONS_100
               MILIMETER : Bool;   // NC AXES PBS LEDS MILIMETER
               SP0_4 : Bool;
               SP0_5 : Bool;
               SP0_6 : Bool;
               SP0_7 : Bool;
               SP1_0 : Bool;
               SP1_1 : Bool;
               SP1_2 : Bool;
               SP1_3 : Bool;
               SP1_4 : Bool;
               SP1_5 : Bool;
               SP1_6 : Bool;
               SP1_7 : Bool;
            END_STRUCT;
         END_STRUCT;
         BA3 : Struct
            SOFTKEYS : Struct   // BA3 SOFTKEYS
               AUTOMATIC_MODE : Bool;   // AUTOMATIC MODE (BA3) / BA3 SOFTKEYS AUTOMATIC MODE
               SINGLE_MODE : Bool;   // SINGLE CYCLE MODE (BA3) / BA3 SOFTKEYS SINGLE MODE
               SEMIAUTOMATIC_MODE : Bool;   // SEMIAUTOMATIC MODE (BA3) / BA3 SOFTKEYS SEMIAUTOMATIC MODE
               MANUAL_MODE : Bool;   // MANUAL MODE (BA3) / BA3 SOFTKEYS MANUAL MODE
               START : Bool;   // START (BA3) / BA3 SOFTKEYS START
               STOP : Bool;   // STOP (BA3) / BA3 SOFTKEYS STOP
               SPARE_2 : Bool;   // BA3 SOFTKEYS SP0 6
               SPARE : Bool;   // BA3 SOFTKEYS SP0 7
               SET_GOOD_PART : Bool;   // BA3 SOFTKEYS CLAMP FIXTURE 1
               UNCLAMP_F1 : Bool;   // BA3 SOFTKEYS UNCLAMP FIXTURE 1
               CLAMP_F2 : Bool;   // BA3 SOFTKEYS CLAMP FIXTURE 2
               UNCLAMP_F2 : Bool;   // BA3 SOFTKEYS UNCLAMP FIXTURE 2
               UNBLOCK_DEVICE : Bool;   // BA3 SOFTKEYS UNBLOCK DEVICE
               HOME : Bool;   // HOME (BA3) / BA3 SOFTKEYS HOME
               END_OF_CYCLE : Bool;   // BA3 SOFTKEYS END OF CYCLE
               CHANGE_PANEL_CONTROL : Bool;   // BA3 SOFTKEYS CHANGE PANEL
            END_STRUCT;
            PBS : Struct   // BA3 PBS
               MICRON : Bool;   // BA3 PBS MICRON
               MICRONS_10 : Bool;   // BA3 PBS MICRONS_10
               MICRONS_100 : Bool;   // BA3 PBS MICRONS_100
               MILIMETER : Bool;   // BA3 PBS MILIMETER
               SP0_4 : Bool;
               SP0_5 : Bool;
               SP0_6 : Bool;
               SP0_7 : Bool;
               SP1_0 : Bool;
               SP1_1 : Bool;
               SP1_2 : Bool;
               SP1_3 : Bool;
               SP1_4 : Bool;
               SP1_5 : Bool;
               SP1_6 : Bool;
               SP1_7 : Bool;
            END_STRUCT;
            SOFTKEY_LEDS : Struct   // BA3 SOFTKEY LEDS
               ER_MODE : Bool;   // BA3 SOFTKEY LEDS ER MODE
               ES_MODE : Bool;   // BA3 SOFTKEY LEDS ES MODE
               HOME : Bool;   // BA3 SOFTKEY LEDS HOME
               START : Bool;   // BA3 SOFTKEY LEDS START
               STOP : Bool;   // BA3 SOFTKEY LEDS STOP
               CONTINUOS_INCREMENTAL : Bool;   // BA3 SOFTKEY LEDS CONTINUOS INCREMENTAL
               SP0_6 : Bool;   // BA3 SOFTKEY LEDS SP0 6
               SP0_7 : Bool;   // BA3 SOFTKEY LEDS SP0 7
               JOG_PLUS : Bool;   // BA3 SOFTKEY LEDS JOG PLUS
               JOG_MINUS : Bool;   // BA3 SOFTKEY LEDS JOG MINUS
               UNBLOCK_DEVICE : Bool;   // BA3 SOFTKEY LEDS UNBLOCK DEVICE
               CLAMP_F1 : Bool;   // BA3 SOFTKEY LEDS CLAMP F1
               UNCLAMP_F1 : Bool;   // BA3 SOFTKEY LEDS UNCLAMP F1
               CLAMP_F2 : Bool;   // BA3 SOFTKEY LEDS CLAMP F2
               UNCLAMP_F2 : Bool;   // BA3 SOFTKEY LEDS UNCLAMP F2
               SP1_7 : Bool;   // BA3 SOFTKEY LEDS SP1 7
            END_STRUCT;
            PBS_LEDS : Struct   // BA3 PBS LEDS
               MICRON : Bool;   // BA3 PBS LEDS MICRON
               MICRONS_10 : Bool;   // BA3 PBS LEDS MICRONS_10
               MICRONS_100 : Bool;   // BA3 PBS LEDS MICRONS_100
               MILIMETER : Bool;   // BA3 PBS LEDS MILIMETER
               SP0_4 : Bool;
               SP0_5 : Bool;
               SP0_6 : Bool;
               SP0_7 : Bool;
               SP1_0 : Bool;
               SP1_1 : Bool;
               SP1_2 : Bool;
               SP1_3 : Bool;
               SP1_4 : Bool;
               SP1_5 : Bool;
               SP1_6 : Bool;
               BA3_MODE_SELECTED : Bool;
            END_STRUCT;
         END_STRUCT;
         AXIS_SELECTED : Struct
            AXIS_1_SELECTED : Bool;   // SPINDLE SP11 SELECTED / AXIS 1 SELECTED
            AXIS_2_SELECTED : Bool;   // SPINDLE SP12 SELECTED / AXIS 2 SELECTED
            AXIS_3_SELECTED : Bool;   // SPINDLE SP13 SELECTED / AXIS 3 SELECTED
            AXIS_4_SELECTED : Bool;   // SPINDLE SP14 SELECTED / AXIS 4 SELECTED
            AXIS_5_SELECTED : Bool;   // AXIS X1 SELECTED / AXIS 5 SELECTED
            AXIS_6_SELECTED : Bool;   // AXIS Y1 SELECTED / AXIS 6 SELECTED
            AXIS_7_SELECTED : Bool;   // AXIS Z11 SELECTED / AXIS 7 SELECTED
            AXIS_8_SELECTED : Bool;   // AXIS Z12 SELECTED / AXIS 8 SELECTED
            AXIS_9_SELECTED : Bool;   // AXIS X2 SELECTED / AXIS 9 SELECTED
            AXIS_10_SELECTED : Bool;   // AXIS Y2 SELECTED / AXIS 10 SELECTED
            AXIS_11_SELECTED : Bool;   // AXIS Z21 SELECTED / AXIS 11 SELECTED
            AXIS_12_SELECTED : Bool;   // AXIS Z22 SELECTED / AXIS 12 SELECTED
            AXIS_13_SELECTED : Bool;   // AXIS Q1 SELECTED / AXIS 13 SELECTED
            AXIS_14_SELECTED : Bool;   // AXIS Q2 SELECTED / AXIS 14 SELECTED
            AXIS_15_SELECTED : Bool;   // AXIS A1 SELECTED / AXIS 15 SELECTED
            AXIS_16_SELECTED : Bool;   // AXIS B SELECTED / AXIS 16 SELECTED
            AXIS_17_SELECTED : Bool;   // AXIS W SELECTED / AXIS 17 SELECTED
            AXIS_18_SELECTED : Bool;   // AXIS E SELECTED / AXIS 18 SELECTED
            AXIS_19_SELECTED : Bool;   // AXIS A2 SELECTED / AXIS 19 SELECTED
            AXIS_20_SELECTED : Bool;   // AXIS V1 SELECTED / AXIS 20 SELECTED
            AXIS_21_SELECTED : Bool;   // AXIS V2 SELECTED / AXIS 21 SELECTED
            AXIS_22_SELECTED : Bool;   // AXIS R SELECTED / AXIS 22 SELECTED
            AXIS_23_SELECTED : Bool;   // AXIS U1 SELECTED / AXIS 23 SELECTED
            AXIS_24_SELECTED : Bool;   // AXIS U2 SELECTED / AXIS 24 SELECTED
            AXIS_25_SELECTED : Bool;   // AXIS C SELECTED / AXIS 25 SELECTED
            AXIS_26_SELECTED : Bool;   // AXIS W1 SELECTED / AXIS 26 SELECTED
            AXIS_27_SELECTED : Bool;   // AXIS V SELECTED / AXIS 27 SELECTED
            AXIS_28_SELECTED : Bool;   // AXIS 28 SELECTED
            AXIS_29_SELECTED : Bool;   // AXIS 29 SELECTED
            AXIS_30_SELECTED : Bool;   // AXIS 30 SELECTED
            AXIS_31_SELECTED : Bool;   // AXIS 31 SELECTED
            SPARE_33_7 : Bool;   // SPARE_33_7
         END_STRUCT;
         AXIS_REFERENCED : Struct
            AXIS_1_REFERENCED : Bool;   // SPINDLE SP11 REFERENCED / AXIS 1 REFERENCED
            AXIS_2_REFERENCED : Bool;   // SPINDLE SP12 REFERENCED / AXIS 2 REFERENCED
            AXIS_3_REFERENCED : Bool;   // SPINDLE SP13 REFERENCED / AXIS 3 REFERENCED
            AXIS_4_REFERENCED : Bool;   // SPINDLE SP14 REFERENCED / AXIS 4 REFERENCED
            AXIS_5_REFERENCED : Bool;   // AXIS X1 REFERENCED / AXIS 5 REFERENCED
            AXIS_6_REFERENCED : Bool;   // AXIS Y1 REFERENCED / AXIS 6 REFERENCED
            AXIS_7_REFERENCED : Bool;   // AXIS Z11 REFERENCED / AXIS 7 REFERENCED
            AXIS_8_REFERENCED : Bool;   // AXIS Z12 REFERENCED / AXIS 8 REFERENCED
            AXIS_9_REFERENCED : Bool;   // AXIS X2 REFERENCED / AXIS 9 REFERENCED
            AXIS_10_REFERENCED : Bool;   // AXIS Y2 REFERENCED / AXIS 10 REFERENCED
            AXIS_11_REFERENCED : Bool;   // AXIS Z21 REFERENCED / AXIS 11 REFERENCED
            AXIS_12_REFERENCED : Bool;   // AXIS Z22 REFERENCED / AXIS 12 REFERENCED
            AXIS_13_REFERENCED : Bool;   // AXIS Q1 REFERENCED / AXIS 13 REFERENCED
            AXIS_14_REFERENCED : Bool;   // AXIS Q2 REFERENCED / AXIS 14 REFERENCED
            AXIS_15_REFERENCED : Bool;   // AXIS A1 REFERENCED / AXIS 15 REFERENCED
            AXIS_16_REFERENCED : Bool;   // AXIS B REFERENCED / AXIS 16 REFERENCED
            AXIS_17_REFERENCED : Bool;   // AXIS W REFERENCED / AXIS 17 REFERENCED
            AXIS_18_REFERENCED : Bool;   // AXIS E REFERENCED / AXIS 18 REFERENCED
            AXIS_19_REFERENCED : Bool;   // AXIS A2 REFERENCED / AXIS 19 REFERENCED
            AXIS_20_REFERENCED : Bool;   // AXIS V1 REFERENCED / AXIS 20 REFERENCED
            AXIS_21_REFERENCED : Bool;   // AXIS V2 REFERENCED / AXIS 21 REFERENCED
            AXIS_22_REFERENCED : Bool;   // AXIS R REFERENCED / AXIS 22 REFERENCED
            AXIS_23_REFERENCED : Bool;   // AXIS U1 REFERENCED / AXIS 23 REFERENCED
            AXIS_24_REFERENCED : Bool;   // AXIS U2 REFERENCED / AXIS 24 REFERENCED
            AXIS_25_REFERENCED : Bool;   // AXIS C REFERENCED / AXIS 25 REFERENCED
            AXIS_26_REFERENCED : Bool;   // AXIS W1 REFERENCED / AXIS 26 REFERENCED
            AXIS_27_REFERENCED : Bool;   // AXIS V REFERENCED / AXIS 27 REFERENCED
            AXIS_28_REFERENCED : Bool;   // AXIS 28 REFERENCED
            AXIS_29_REFERENCED : Bool;   // AXIS 29 REFERENCED
            AXIS_30_REFERENCED : Bool;   // AXIS 30 REFERENCED
            AXIS_31_REFERENCED : Bool;   // AXIS 31 REFERENCED
            SPARE_37_7 : Bool;   // SPARE_37_7
         END_STRUCT;
         AXIS_CONDITIONS : Struct
            AXIS_1_CONDITIONS : Bool;   // SPINDLE SP11 CONDITIONS / AXIS 1 CONDITIONS
            AXIS_2_CONDITIONS : Bool;   // SPINDLE SP12 CONDITIONS / AXIS 2 CONDITIONS
            AXIS_3_CONDITIONS : Bool;   // SPINDLE SP13 CONDITIONS / AXIS 3 CONDITIONS
            AXIS_4_CONDITIONS : Bool;   // SPINDLE SP14 CONDITIONS / AXIS 4 CONDITIONS
            AXIS_5_CONDITIONS : Bool;   // AXIS X1 CONDITIONS / AXIS 5 CONDITIONS
            AXIS_6_CONDITIONS : Bool;   // AXIS Y1 CONDITIONS / AXIS 6 CONDITIONS
            AXIS_7_CONDITIONS : Bool;   // AXIS Z11 CONDITIONS / AXIS 7 CONDITIONS
            AXIS_8_CONDITIONS : Bool;   // AXIS Z12 CONDITIONS / AXIS 8 CONDITIONS
            AXIS_9_CONDITIONS : Bool;   // AXIS X2 CONDITIONS / AXIS 9 CONDITIONS
            AXIS_10_CONDITIONS : Bool;   // AXIS Y2 CONDITIONS / AXIS 10 CONDITIONS
            AXIS_11_CONDITIONS : Bool;   // AXIS Z21 CONDITIONS / AXIS 11 CONDITIONS
            AXIS_12_CONDITIONS : Bool;   // AXIS Z22 CONDITIONS / AXIS 12 CONDITIONS
            AXIS_13_CONDITIONS : Bool;   // AXIS Q1 CONDITIONS / AXIS 13 CONDITIONS
            AXIS_14_CONDITIONS : Bool;   // AXIS Q2 CONDITIONS / AXIS 14 CONDITIONS
            AXIS_15_CONDITIONS : Bool;   // AXIS A1 CONDITIONS / AXIS 15 CONDITIONS
            AXIS_16_CONDITIONS : Bool;   // AXIS B CONDITIONS / AXIS 16 CONDITIONS
            AXIS_17_CONDITIONS : Bool;   // AXIS W CONDITIONS / AXIS 17 CONDITIONS
            AXIS_18_CONDITIONS : Bool;   // AXIS E CONDITIONS / AXIS 18 CONDITIONS
            AXIS_19_CONDITIONS : Bool;   // AXIS A2 CONDITIONS / AXIS 19 CONDITIONS
            AXIS_20_CONDITIONS : Bool;   // AXIS V1 CONDITIONS / AXIS 20 CONDITIONS
            AXIS_21_CONDITIONS : Bool;   // AXIS V2 CONDITIONS / AXIS 21 CONDITIONS
            AXIS_22_CONDITIONS : Bool;   // AXIS R CONDITIONS / AXIS 22 CONDITIONS
            AXIS_23_CONDITIONS : Bool;   // AXIS U1 CONDITIONS / AXIS 23 CONDITIONS
            AXIS_24_CONDITIONS : Bool;   // AXIS U2 CONDITIONS / AXIS 24 CONDITIONS
            AXIS_25_CONDITIONS : Bool;   // AXIS C CONDITIONS / AXIS 25 CONDITIONS
            AXIS_26_CONDITIONS : Bool;   // AXIS W1 CONDITIONS / AXIS 26 CONDITIONS
            AXIS_27_CONDITIONS : Bool;   // AXIS V CONDITIONS / AXIS 27 CONDITIONS
            AXIS_28_CONDITIONS : Bool;   // AXIS 28 CONDITIONS
            AXIS_29_CONDITIONS : Bool;   // AXIS 29 CONDITIONS
            AXIS_30_CONDITIONS : Bool;   // AXIS 30 CONDITIONS
            AXIS_31_CONDITIONS : Bool;   // AXIS 31 CONDITIONS
            SPARE_41_7 : Bool;   // SPARE_41_7
         END_STRUCT;
         AXIS_POSITION : Struct
            AXIS_1_POSITION : Real;   // AXIS 1 POSITION
            AXIS_2_POSITION : Real;   // AXIS 2 POSITION
            AXIS_3_POSITION : Real;   // AXIS 3 POSITION
            AXIS_4_POSITION : Real;   // AXIS 4 POSITION
            AXIS_5_POSITION : Real;   // AXIS 5 POSITION
            AXIS_6_POSITION : Real;   // AXIS 6 POSITION
            AXIS_7_POSITION : Real;   // AXIS 7 POSITION
            AXIS_8_POSITION : Real;   // AXIS 8 POSITION
            AXIS_9_POSITION : Real;   // AXIS 9 POSITION
            AXIS_10_POSITION : Real;   // AXIS 10 POSITION
            AXIS_11_POSITION : Real;   // AXIS 11 POSITION
            AXIS_12_POSITION : Real;   // AXIS 12 POSITION
            AXIS_13_POSITION : Real;   // AXIS 13 POSITION
            AXIS_14_POSITION : Real;   // AXIS 14 POSITION
            AXIS_15_POSITION : Real;   // AXIS 15 POSITION
            AXIS_16_POSITION : Real;   // AXIS 16 POSITION
            AXIS_17_POSITION : Real;   // AXIS 17 POSITION
            AXIS_18_POSITION : Real;   // AXIS 18 POSITION
            AXIS_19_POSITION : Real;   // AXIS 19 POSITION
            AXIS_20_POSITION : Real;   // AXIS 20 POSITION
            AXIS_21_POSITION : Real;   // AXIS 21 POSITION
            AXIS_22_POSITION : Real;   // AXIS 22 POSITION
            AXIS_23_POSITION : Real;   // AXIS 23 POSITION
            AXIS_24_POSITION : Real;   // AXIS 24 POSITION
            AXIS_25_POSITION : Real;   // AXIS 25 POSITION
            AXIS_26_POSITION : Real;   // AXIS 26 POSITION
            AXIS_27_POSITION : Real;   // AXIS 27 POSITION
            AXIS_28_POSITION : Real;   // AXIS 28 POSITION
            AXIS_29_POSITION : Real;   // AXIS 29 POSITION
            AXIS_30_POSITION : Real;   // AXIS 30 POSITION
            AXIS_31_POSITION : Real;   // AXIS 31 POSITION
         END_STRUCT;
         AUX : Struct
            AUX1 : Bool;   // AUXILIAR 1
            AUX2 : Bool;   // AUXILIAR 2
            AUX3 : Bool;   // AUXILIAR 3
            AUX4 : Bool;   // AUXILIAR 4
            AUX5 : Bool;   // AUXILIAR 5
            AUX6 : Bool;   // AUXILIAR 6
            AUX7 : Bool;   // AUXILIAR 7
            AUX8 : Byte;   // AUXILIAR 8
            AUX9 : Byte;   // AUXILIAR 9
            AUX10 : Byte;   // AUXILIAR 10
            AUX11 : Byte;   // AUXILIAR 11
            AUX12 : Byte;   // AUXILIAR 12
            AUX13 : Byte;   // AUXILIAR 13
            AUX14 : Byte;   // AUXILIAR 14
         END_STRUCT;
         REFERENCE_SCREEN : Struct
            AXIS_SELECTED : Int;   // REFERENCE SCREEN AXIS SELECTED
            MEMO_AXIS_SELECTED : Int;   // REFERENCE SCREEN MEMORIZED AXIS SELECTED
            SCREEN_SELECTED : Bool;   // REFERENCE SCREEN SCREEN SELECTED
            READ_DATA : Bool;   // REFERENCE SCREEN READ DATA
            WRITE_DATA : Bool;   // REFERENCE SCREEN WRITE DATA
            TIMER_READ : TP_TIME;   // READ TIMER
         END_STRUCT;
      END_STRUCT;
      MG10 : Struct
         GENERAL_BITS : Struct
            SCREEN_BA3_SELECTED : Bool;   // SCREEN BA3 SELECTED / GENERAL BITS SCREEN BA3 SELECTED
            SCREEN_NC_MANUAL_SELECTED : Bool;   // SCREEN NC MANUAL SELECTED / GENERAL BITS SCREEN NC MANUAL SELECTED
            SCREEN_EB_MODE_SELECT : Bool;   // SCREEN EB MODE SELECT / GENERAL BITS SCREEN EB MODE SELECT
            SP0_3 : Bool;   // GENERAL BITS
            BA3_SELECTED_UNIT_1 : Bool;   // BA3 SELECTED UNIT 1 / GENERAL BITS BA3 LIST SELECTED UNIT 1
            BA3_SELECTED_UNIT_2 : Bool;   // BA3 SELECTED UNIT 2 / GENERAL BITS BA3 LIST SELECTED UNIT 2
            BA3_SELECTED_UNIT_3 : Bool;   // BA3 SELECTED UNIT 3 / GENERAL BITS BA3 LIST SELECTED UNIT 3
            BA3_SELECTED_UNIT_4 : Bool;   // BA3 SELECTED UNIT 4 / GENERAL BITS BA3 LIST SELECTED UNIT 4
            SP1_0 : Bool;   // TWO UNITS OPTION ENABLE / GENERAL BITS
            SPNDLS_SBH_SG_AUX : Bool;   // GENERAL BITS SPINDLES SBH SG AUX
            SPNDLS_SBH_SG_PULSE : Bool;   // GENERAL BITS SPINDLES SBH SG PULSE
            PLC_LINE_AXES_BYTE : Byte;   // GENERAL BITS PLC LINE AXES BYTE
            PLC_LINE_SPINDLES_BYTE : Byte;   // GENERAL BITS PLC LINE SPINDLES BYTE
            PLC_LINE_AXES : Int;   // GENERAL BITS PLC LINE AXES
            PLC_LINE_SPINDLES : Int;   // GENERAL BITS PLC LINE SPINDLES
            BA3_LIST : Int;   // GENERAL BITS BA3 LIST
            MINUS_KEY : Byte;   // GENERAL BITS MINUS KEY
            PLUS_KEY : Byte;   // GENERAL BITS PLUS KEY
         END_STRUCT;
         NC_AXES : Struct
            SOFTKEYS : Struct   // NC AXES SOFTKEYS
               LEFT : Struct
                  MANUAL_MODE : Bool;   // MANUAL MODE (CN-AXES SCREEN) / NC AXES SOFTKEYS MANUAL MODE
                  SEMIAUTOMATIC_MODE : Bool;   // SEMIAUTOMATIC MODE (CN-AXES SCREEN) / NC AXES SOFTKEYS SEMIAUTOMATIC MODE
                  REFERENCE_MODE : Bool;   // REFERENCE MODE (CN-AXES SCREEN) / NC AXES SOFTKEYS REFERENCE MODE
                  JOG_MODE : Bool;   // NC AXES SOFTKEYS SPARE
                  SPINDLES_SBH_SG : Bool;   // SPINDLES SBH SG (CN-AXES SCREEN) / NC AXES SOFTKEYS SPINDLES SBH SG
                  CONTINUOS_INCREMENTAL : Bool;   // CONTINUOS-INCREMENTAL (CN-AXES SCREEN) / NC AXES SOFTKEYS CONTINUOS INCREMENTAL
                  SP0_6 : Bool;   // NC AXES SOFTKEYS SP0 6
                  SP0_7 : Bool;   // NC AXES SOFTKEYS SP0 7
               END_STRUCT;
               RIGHT : Struct
                  JOG_PLUS : Bool;   // JOG PLUS (CN-AXES SCREEN) / NC AXES SOFTKEYS JOG PLUS
                  JOG_MINUS : Bool;   // JOG MINUS (CN-AXES SCREEN) / NC AXES SOFTKEYS JOG MINUS
                  BLOCK_DEVICE : Bool;   // BLOCK DEVICE (CN-AXES SCREEN) / NC AXES SOFTKEYS BLOCK DEVICE
                  UNBLOCK_DEVICE : Bool;   // UNBLOCK DEVICE (CN-AXES SCREEN) / NC AXES SOFTKEYS UNBLOCK DEVICE
                  SP1_4 : Bool;   // NC AXES SOFTKEYS SP1 4
                  CHANGE_PANEL_CONTROL : Bool;   // CHANGE PANEL CONTROL (CN-AXES SCREEN) / NC AXES SOFTKEYS CHANGE PANEL CONTROL
                  SP1_6 : Bool;   // NC AXES SOFTKEYS SP1 6
                  SP1_7 : Bool;   // NC AXES SOFTKEYS SP1 7
               END_STRUCT;
            END_STRUCT;
            PBS : Struct   // NC AXES PBS
               MICRON : Bool;   // NC AXES PBS MICRON
               MICRONS_10 : Bool;   // NC AXES PBS MICRONS 10
               MICRONS_100 : Bool;   // NC AXES PBS MICRONS 100
               MILIMETER : Bool;   // NC AXES PBS MILIMETER
               SP0_4 : Bool;
               SP0_5 : Bool;
               SP0_6 : Bool;
               SP0_7 : Bool;
               SP1_0 : Bool;
               SP1_1 : Bool;
               SP1_2 : Bool;
               SP1_3 : Bool;
               SP1_4 : Bool;
               SP1_5 : Bool;
               SP1_6 : Bool;
               SP1_7 : Bool;
            END_STRUCT;
            SOFTKEY_LEDS : Struct   // NC AXES SOFTKEY LEDS
               MANUAL_MODE : Bool;   // MANUAL MODE (SOFTKEY LEDS) / NC AXES SOFTKEY LEDS MANUAL MODE
               ES_MODE : Bool;   // NC AXES SOFTKEY LEDS ES MODE
               REFERENCE_MODE : Bool;   // NC AXES SOFTKEY LEDS REFERENCE MODE
               SP0_3 : Bool;   // NC AXES SOFTKEY LEDS SP0 3
               SPINDLES_SBH_SG : Bool;   // NC AXES SOFTKEY LEDS SPINDLES SBH SG
               CONTINUOS_INCREMENTAL : Bool;   // NC AXES SOFTKEY LEDS CONTINUOS INCREMENTAL
               EB_MODE : Bool;   // NC AXES SOFTKEY LEDS EB MODE
               VK_MODE : Bool;   // NC AXES SOFTKEY LEDS VK MODE
               JOG_PLUS : Bool;   // NC AXES SOFTKEY LEDS JOG PLUS
               JOG_MINUS : Bool;   // NC AXES SOFTKEY LEDS JOG MINUS
               BLOCK_DEVICE : Bool;   // NC AXES SOFTKEY LEDS BLOCK DEVICE
               UNBLOCK_DEVICE : Bool;   // NC AXES SOFTKEY LEDS UNBLOCK DEVICE
               SP1_4 : Bool;   // NC AXES SOFTKEY LEDS SP1 4
               CHANGE_PANEL_CONTROL : Bool;   // NC AXES SOFTKEY LEDS CHANGE PANEL CONTROL
               SP1_6 : Bool;   // NC AXES SOFTKEY LEDS SP1 6
               SP1_7 : Bool;   // NC AXES SOFTKEY LEDS SP1 7
            END_STRUCT;
            PBS_LEDS : Struct   // NC AXES PBS LEDS
               MICRON : Bool;   // NC AXES PBS LEDS MICRON
               MICRONS_10 : Bool;   // NC AXES PBS LEDS MICRONS_10
               MICRONS_100 : Bool;   // NC AXES PBS LEDS MICRONS_100
               MILIMETER : Bool;   // NC AXES PBS LEDS MILIMETER
               SP0_4 : Bool;
               SP0_5 : Bool;
               SP0_6 : Bool;
               SP0_7 : Bool;
               SP1_0 : Bool;
               SP1_1 : Bool;
               SP1_2 : Bool;
               SP1_3 : Bool;
               SP1_4 : Bool;
               SP1_5 : Bool;
               SP1_6 : Bool;
               SP1_7 : Bool;
            END_STRUCT;
         END_STRUCT;
         BA3 : Struct
            SOFTKEYS : Struct   // BA3 SOFTKEYS
               AUTOMATIC_MODE : Bool;   // AUTOMATIC MODE (BA3) / BA3 SOFTKEYS AUTOMATIC MODE
               SINGLE_MODE : Bool;   // SINGLE CYCLE MODE (BA3) / BA3 SOFTKEYS SINGLE MODE
               SEMIAUTOMATIC_MODE : Bool;   // SEMIAUTOMATIC MODE (BA3) / BA3 SOFTKEYS SEMIAUTOMATIC MODE
               MANUAL_MODE : Bool;   // MANUAL MODE (BA3) / BA3 SOFTKEYS MANUAL MODE
               START : Bool;   // START (BA3) / BA3 SOFTKEYS START
               STOP : Bool;   // STOP (BA3) / BA3 SOFTKEYS STOP
               SPARE_2 : Bool;   // BA3 SOFTKEYS SP0 6
               SPARE : Bool;   // BA3 SOFTKEYS SP0 7
               SET_GOOD_PART : Bool;   // BA3 SOFTKEYS CLAMP FIXTURE 1
               UNCLAMP_F1 : Bool;   // BA3 SOFTKEYS UNCLAMP FIXTURE 1
               CLAMP_F2 : Bool;   // BA3 SOFTKEYS CLAMP FIXTURE 2
               UNCLAMP_F2 : Bool;   // BA3 SOFTKEYS UNCLAMP FIXTURE 2
               UNBLOCK_DEVICE : Bool;   // BA3 SOFTKEYS UNBLOCK DEVICE
               HOME : Bool;   // HOME (BA3) / BA3 SOFTKEYS HOME
               END_OF_CYCLE : Bool;   // BA3 SOFTKEYS END OF CYCLE
               CHANGE_PANEL_CONTROL : Bool;   // BA3 SOFTKEYS CHANGE PANEL
            END_STRUCT;
            PBS : Struct   // BA3 PBS
               MICRON : Bool;   // BA3 PBS MICRON
               MICRONS_10 : Bool;   // BA3 PBS MICRONS_10
               MICRONS_100 : Bool;   // BA3 PBS MICRONS_100
               MILIMETER : Bool;   // BA3 PBS MILIMETER
               SP0_4 : Bool;
               SP0_5 : Bool;
               SP0_6 : Bool;
               SP0_7 : Bool;
               SP1_0 : Bool;
               SP1_1 : Bool;
               SP1_2 : Bool;
               SP1_3 : Bool;
               SP1_4 : Bool;
               SP1_5 : Bool;
               SP1_6 : Bool;
               SP1_7 : Bool;
            END_STRUCT;
            SOFTKEY_LEDS : Struct   // BA3 SOFTKEY LEDS
               ER_MODE : Bool;   // BA3 SOFTKEY LEDS ER MODE
               ES_MODE : Bool;   // BA3 SOFTKEY LEDS ES MODE
               HOME : Bool;   // BA3 SOFTKEY LEDS HOME
               START : Bool;   // BA3 SOFTKEY LEDS START
               STOP : Bool;   // BA3 SOFTKEY LEDS STOP
               CONTINUOS_INCREMENTAL : Bool;   // BA3 SOFTKEY LEDS CONTINUOS INCREMENTAL
               SP0_6 : Bool;   // BA3 SOFTKEY LEDS SP0 6
               SP0_7 : Bool;   // BA3 SOFTKEY LEDS SP0 7
               JOG_PLUS : Bool;   // BA3 SOFTKEY LEDS JOG PLUS
               JOG_MINUS : Bool;   // BA3 SOFTKEY LEDS JOG MINUS
               UNBLOCK_DEVICE : Bool;   // BA3 SOFTKEY LEDS UNBLOCK DEVICE
               CLAMP_F1 : Bool;   // BA3 SOFTKEY LEDS CLAMP F1
               UNCLAMP_F1 : Bool;   // BA3 SOFTKEY LEDS UNCLAMP F1
               CLAMP_F2 : Bool;   // BA3 SOFTKEY LEDS CLAMP F2
               UNCLAMP_F2 : Bool;   // BA3 SOFTKEY LEDS UNCLAMP F2
               SP1_7 : Bool;   // BA3 SOFTKEY LEDS SP1 7
            END_STRUCT;
            PBS_LEDS : Struct   // BA3 PBS LEDS
               MICRON : Bool;   // BA3 PBS LEDS MICRON
               MICRONS_10 : Bool;   // BA3 PBS LEDS MICRONS_10
               MICRONS_100 : Bool;   // BA3 PBS LEDS MICRONS_100
               MILIMETER : Bool;   // BA3 PBS LEDS MILIMETER
               SP0_4 : Bool;
               SP0_5 : Bool;
               SP0_6 : Bool;
               SP0_7 : Bool;
               SP1_0 : Bool;
               SP1_1 : Bool;
               SP1_2 : Bool;
               SP1_3 : Bool;
               SP1_4 : Bool;
               SP1_5 : Bool;
               SP1_6 : Bool;
               BA3_MODE_SELECTED : Bool;
            END_STRUCT;
         END_STRUCT;
         AXIS_SELECTED : Struct
            AXIS_1_SELECTED : Bool;   // SPINDLE SP11 SELECTED / AXIS 1 SELECTED
            AXIS_2_SELECTED : Bool;   // SPINDLE SP12 SELECTED / AXIS 2 SELECTED
            AXIS_3_SELECTED : Bool;   // SPINDLE SP13 SELECTED / AXIS 3 SELECTED
            AXIS_4_SELECTED : Bool;   // SPINDLE SP14 SELECTED / AXIS 4 SELECTED
            AXIS_5_SELECTED : Bool;   // AXIS X1 SELECTED / AXIS 5 SELECTED
            AXIS_6_SELECTED : Bool;   // AXIS Y1 SELECTED / AXIS 6 SELECTED
            AXIS_7_SELECTED : Bool;   // AXIS Z11 SELECTED / AXIS 7 SELECTED
            AXIS_8_SELECTED : Bool;   // AXIS Z12 SELECTED / AXIS 8 SELECTED
            AXIS_9_SELECTED : Bool;   // AXIS X2 SELECTED / AXIS 9 SELECTED
            AXIS_10_SELECTED : Bool;   // AXIS Y2 SELECTED / AXIS 10 SELECTED
            AXIS_11_SELECTED : Bool;   // AXIS Z21 SELECTED / AXIS 11 SELECTED
            AXIS_12_SELECTED : Bool;   // AXIS Z22 SELECTED / AXIS 12 SELECTED
            AXIS_13_SELECTED : Bool;   // AXIS Q1 SELECTED / AXIS 13 SELECTED
            AXIS_14_SELECTED : Bool;   // AXIS Q2 SELECTED / AXIS 14 SELECTED
            AXIS_15_SELECTED : Bool;   // AXIS A1 SELECTED / AXIS 15 SELECTED
            AXIS_16_SELECTED : Bool;   // AXIS B SELECTED / AXIS 16 SELECTED
            AXIS_17_SELECTED : Bool;   // AXIS W SELECTED / AXIS 17 SELECTED
            AXIS_18_SELECTED : Bool;   // AXIS E SELECTED / AXIS 18 SELECTED
            AXIS_19_SELECTED : Bool;   // AXIS A2 SELECTED / AXIS 19 SELECTED
            AXIS_20_SELECTED : Bool;   // AXIS V1 SELECTED / AXIS 20 SELECTED
            AXIS_21_SELECTED : Bool;   // AXIS V2 SELECTED / AXIS 21 SELECTED
            AXIS_22_SELECTED : Bool;   // AXIS R SELECTED / AXIS 22 SELECTED
            AXIS_23_SELECTED : Bool;   // AXIS U1 SELECTED / AXIS 23 SELECTED
            AXIS_24_SELECTED : Bool;   // AXIS U2 SELECTED / AXIS 24 SELECTED
            AXIS_25_SELECTED : Bool;   // AXIS C SELECTED / AXIS 25 SELECTED
            AXIS_26_SELECTED : Bool;   // AXIS W1 SELECTED / AXIS 26 SELECTED
            AXIS_27_SELECTED : Bool;   // AXIS V SELECTED / AXIS 27 SELECTED
            AXIS_28_SELECTED : Bool;   // AXIS 28 SELECTED
            AXIS_29_SELECTED : Bool;   // AXIS 29 SELECTED
            AXIS_30_SELECTED : Bool;   // AXIS 30 SELECTED
            AXIS_31_SELECTED : Bool;   // AXIS 31 SELECTED
            SPARE_33_7 : Bool;   // SPARE_33_7
         END_STRUCT;
         AXIS_REFERENCED : Struct
            AXIS_1_REFERENCED : Bool;   // SPINDLE SP11 REFERENCED / AXIS 1 REFERENCED
            AXIS_2_REFERENCED : Bool;   // SPINDLE SP12 REFERENCED / AXIS 2 REFERENCED
            AXIS_3_REFERENCED : Bool;   // SPINDLE SP13 REFERENCED / AXIS 3 REFERENCED
            AXIS_4_REFERENCED : Bool;   // SPINDLE SP14 REFERENCED / AXIS 4 REFERENCED
            AXIS_5_REFERENCED : Bool;   // AXIS X1 REFERENCED / AXIS 5 REFERENCED
            AXIS_6_REFERENCED : Bool;   // AXIS Y1 REFERENCED / AXIS 6 REFERENCED
            AXIS_7_REFERENCED : Bool;   // AXIS Z11 REFERENCED / AXIS 7 REFERENCED
            AXIS_8_REFERENCED : Bool;   // AXIS Z12 REFERENCED / AXIS 8 REFERENCED
            AXIS_9_REFERENCED : Bool;   // AXIS X2 REFERENCED / AXIS 9 REFERENCED
            AXIS_10_REFERENCED : Bool;   // AXIS Y2 REFERENCED / AXIS 10 REFERENCED
            AXIS_11_REFERENCED : Bool;   // AXIS Z21 REFERENCED / AXIS 11 REFERENCED
            AXIS_12_REFERENCED : Bool;   // AXIS Z22 REFERENCED / AXIS 12 REFERENCED
            AXIS_13_REFERENCED : Bool;   // AXIS Q1 REFERENCED / AXIS 13 REFERENCED
            AXIS_14_REFERENCED : Bool;   // AXIS Q2 REFERENCED / AXIS 14 REFERENCED
            AXIS_15_REFERENCED : Bool;   // AXIS A1 REFERENCED / AXIS 15 REFERENCED
            AXIS_16_REFERENCED : Bool;   // AXIS B REFERENCED / AXIS 16 REFERENCED
            AXIS_17_REFERENCED : Bool;   // AXIS W REFERENCED / AXIS 17 REFERENCED
            AXIS_18_REFERENCED : Bool;   // AXIS E REFERENCED / AXIS 18 REFERENCED
            AXIS_19_REFERENCED : Bool;   // AXIS A2 REFERENCED / AXIS 19 REFERENCED
            AXIS_20_REFERENCED : Bool;   // AXIS V1 REFERENCED / AXIS 20 REFERENCED
            AXIS_21_REFERENCED : Bool;   // AXIS V2 REFERENCED / AXIS 21 REFERENCED
            AXIS_22_REFERENCED : Bool;   // AXIS R REFERENCED / AXIS 22 REFERENCED
            AXIS_23_REFERENCED : Bool;   // AXIS U1 REFERENCED / AXIS 23 REFERENCED
            AXIS_24_REFERENCED : Bool;   // AXIS U2 REFERENCED / AXIS 24 REFERENCED
            AXIS_25_REFERENCED : Bool;   // AXIS C REFERENCED / AXIS 25 REFERENCED
            AXIS_26_REFERENCED : Bool;   // AXIS W1 REFERENCED / AXIS 26 REFERENCED
            AXIS_27_REFERENCED : Bool;   // AXIS V REFERENCED / AXIS 27 REFERENCED
            AXIS_28_REFERENCED : Bool;   // AXIS 28 REFERENCED
            AXIS_29_REFERENCED : Bool;   // AXIS 29 REFERENCED
            AXIS_30_REFERENCED : Bool;   // AXIS 30 REFERENCED
            AXIS_31_REFERENCED : Bool;   // AXIS 31 REFERENCED
            SPARE_37_7 : Bool;   // SPARE_37_7
         END_STRUCT;
         AXIS_CONDITIONS : Struct
            AXIS_1_CONDITIONS : Bool;   // SPINDLE SP11 CONDITIONS / AXIS 1 CONDITIONS
            AXIS_2_CONDITIONS : Bool;   // SPINDLE SP12 CONDITIONS / AXIS 2 CONDITIONS
            AXIS_3_CONDITIONS : Bool;   // SPINDLE SP13 CONDITIONS / AXIS 3 CONDITIONS
            AXIS_4_CONDITIONS : Bool;   // SPINDLE SP14 CONDITIONS / AXIS 4 CONDITIONS
            AXIS_5_CONDITIONS : Bool;   // AXIS X1 CONDITIONS / AXIS 5 CONDITIONS
            AXIS_6_CONDITIONS : Bool;   // AXIS Y1 CONDITIONS / AXIS 6 CONDITIONS
            AXIS_7_CONDITIONS : Bool;   // AXIS Z11 CONDITIONS / AXIS 7 CONDITIONS
            AXIS_8_CONDITIONS : Bool;   // AXIS Z12 CONDITIONS / AXIS 8 CONDITIONS
            AXIS_9_CONDITIONS : Bool;   // AXIS X2 CONDITIONS / AXIS 9 CONDITIONS
            AXIS_10_CONDITIONS : Bool;   // AXIS Y2 CONDITIONS / AXIS 10 CONDITIONS
            AXIS_11_CONDITIONS : Bool;   // AXIS Z21 CONDITIONS / AXIS 11 CONDITIONS
            AXIS_12_CONDITIONS : Bool;   // AXIS Z22 CONDITIONS / AXIS 12 CONDITIONS
            AXIS_13_CONDITIONS : Bool;   // AXIS Q1 CONDITIONS / AXIS 13 CONDITIONS
            AXIS_14_CONDITIONS : Bool;   // AXIS Q2 CONDITIONS / AXIS 14 CONDITIONS
            AXIS_15_CONDITIONS : Bool;   // AXIS A1 CONDITIONS / AXIS 15 CONDITIONS
            AXIS_16_CONDITIONS : Bool;   // AXIS B CONDITIONS / AXIS 16 CONDITIONS
            AXIS_17_CONDITIONS : Bool;   // AXIS W CONDITIONS / AXIS 17 CONDITIONS
            AXIS_18_CONDITIONS : Bool;   // AXIS E CONDITIONS / AXIS 18 CONDITIONS
            AXIS_19_CONDITIONS : Bool;   // AXIS A2 CONDITIONS / AXIS 19 CONDITIONS
            AXIS_20_CONDITIONS : Bool;   // AXIS V1 CONDITIONS / AXIS 20 CONDITIONS
            AXIS_21_CONDITIONS : Bool;   // AXIS V2 CONDITIONS / AXIS 21 CONDITIONS
            AXIS_22_CONDITIONS : Bool;   // AXIS R CONDITIONS / AXIS 22 CONDITIONS
            AXIS_23_CONDITIONS : Bool;   // AXIS U1 CONDITIONS / AXIS 23 CONDITIONS
            AXIS_24_CONDITIONS : Bool;   // AXIS U2 CONDITIONS / AXIS 24 CONDITIONS
            AXIS_25_CONDITIONS : Bool;   // AXIS C CONDITIONS / AXIS 25 CONDITIONS
            AXIS_26_CONDITIONS : Bool;   // AXIS W1 CONDITIONS / AXIS 26 CONDITIONS
            AXIS_27_CONDITIONS : Bool;   // AXIS V CONDITIONS / AXIS 27 CONDITIONS
            AXIS_28_CONDITIONS : Bool;   // AXIS 28 CONDITIONS
            AXIS_29_CONDITIONS : Bool;   // AXIS 29 CONDITIONS
            AXIS_30_CONDITIONS : Bool;   // AXIS 30 CONDITIONS
            AXIS_31_CONDITIONS : Bool;   // AXIS 31 CONDITIONS
            SPARE_41_7 : Bool;   // SPARE_41_7
         END_STRUCT;
         AXIS_POSITION : Struct
            AXIS_1_POSITION : Real;   // AXIS 1 POSITION
            AXIS_2_POSITION : Real;   // AXIS 2 POSITION
            AXIS_3_POSITION : Real;   // AXIS 3 POSITION
            AXIS_4_POSITION : Real;   // AXIS 4 POSITION
            AXIS_5_POSITION : Real;   // AXIS 5 POSITION
            AXIS_6_POSITION : Real;   // AXIS 6 POSITION
            AXIS_7_POSITION : Real;   // AXIS 7 POSITION
            AXIS_8_POSITION : Real;   // AXIS 8 POSITION
            AXIS_9_POSITION : Real;   // AXIS 9 POSITION
            AXIS_10_POSITION : Real;   // AXIS 10 POSITION
            AXIS_11_POSITION : Real;   // AXIS 11 POSITION
            AXIS_12_POSITION : Real;   // AXIS 12 POSITION
            AXIS_13_POSITION : Real;   // AXIS 13 POSITION
            AXIS_14_POSITION : Real;   // AXIS 14 POSITION
            AXIS_15_POSITION : Real;   // AXIS 15 POSITION
            AXIS_16_POSITION : Real;   // AXIS 16 POSITION
            AXIS_17_POSITION : Real;   // AXIS 17 POSITION
            AXIS_18_POSITION : Real;   // AXIS 18 POSITION
            AXIS_19_POSITION : Real;   // AXIS 19 POSITION
            AXIS_20_POSITION : Real;   // AXIS 20 POSITION
            AXIS_21_POSITION : Real;   // AXIS 21 POSITION
            AXIS_22_POSITION : Real;   // AXIS 22 POSITION
            AXIS_23_POSITION : Real;   // AXIS 23 POSITION
            AXIS_24_POSITION : Real;   // AXIS 24 POSITION
            AXIS_25_POSITION : Real;   // AXIS 25 POSITION
            AXIS_26_POSITION : Real;   // AXIS 26 POSITION
            AXIS_27_POSITION : Real;   // AXIS 27 POSITION
            AXIS_28_POSITION : Real;   // AXIS 28 POSITION
            AXIS_29_POSITION : Real;   // AXIS 29 POSITION
            AXIS_30_POSITION : Real;   // AXIS 30 POSITION
            AXIS_31_POSITION : Real;   // AXIS 31 POSITION
         END_STRUCT;
         AUX : Struct
            AUX1 : Bool;   // AUXILIAR 1
            AUX2 : Bool;   // AUXILIAR 2
            AUX3 : Bool;   // AUXILIAR 3
            AUX4 : Bool;   // AUXILIAR 4
            AUX5 : Bool;   // AUXILIAR 5
            AUX6 : Bool;   // AUXILIAR 6
            AUX7 : Bool;   // AUXILIAR 7
            AUX8 : Byte;   // AUXILIAR 8
            AUX9 : Byte;   // AUXILIAR 9
            AUX10 : Byte;   // AUXILIAR 10
            AUX11 : Byte;   // AUXILIAR 11
            AUX12 : Byte;   // AUXILIAR 12
            AUX13 : Byte;   // AUXILIAR 13
            AUX14 : Byte;   // AUXILIAR 14
         END_STRUCT;
         REFERENCE_SCREEN : Struct
            AXIS_SELECTED : Int;   // REFERENCE SCREEN AXIS SELECTED
            MEMO_AXIS_SELECTED : Int;   // REFERENCE SCREEN MEMORIZED AXIS SELECTED
            SCREEN_SELECTED : Bool;   // REFERENCE SCREEN SCREEN SELECTED
            READ_DATA : Bool;   // REFERENCE SCREEN READ DATA
            WRITE_DATA : Bool;   // REFERENCE SCREEN WRITE DATA
            TIMER_READ : TP_TIME;   // READ TIMER
         END_STRUCT;
      END_STRUCT;
   END_VAR
BEGIN
   MG2.REFERENCE_SCREEN.TIMER_READ.PT := T#500ms;
   MG3.REFERENCE_SCREEN.TIMER_READ.PT := T#500ms;
   MG4.REFERENCE_SCREEN.TIMER_READ.PT := T#500ms;
   MG5.REFERENCE_SCREEN.TIMER_READ.PT := T#500ms;
   MG6.REFERENCE_SCREEN.TIMER_READ.PT := T#500ms;
   MG7.REFERENCE_SCREEN.TIMER_READ.PT := T#500ms;
   MG8.REFERENCE_SCREEN.TIMER_READ.PT := T#500ms;
   MG9.REFERENCE_SCREEN.TIMER_READ.PT := T#500ms;
   MG10.REFERENCE_SCREEN.TIMER_READ.PT := T#500ms;
END_DATA_BLOCK
